// TwinCAT 3 PLC project Xts_Library
// Title: Xts Library
// Company: BeckhoffUK
// Author: ChrisK
// ProjectVersion: 16.0.2
// Description: Xts framework implementation
// ProgramVersion: 3.1.4026.20
// libraries:
//   Base Library, * (Beckhoff UK)
//   Motion Library, * (Beckhoff UK)
//   Tc2_MC2, * (Beckhoff Automation GmbH)
//   Tc2_Standard, * (Beckhoff Automation GmbH)
//   Tc2_System, * (Beckhoff Automation GmbH)
//   Tc3_Mc3Definitions, * (Beckhoff Automation GmbH)
//   Tc3_McCollisionAvoidance, * (Beckhoff Automation GmbH)
//   Tc3_McCoordinatedMotion, * (Beckhoff Automation GmbH)
//   Tc3_Module, * (Beckhoff Automation GmbH)
//   Tc3_XTS_Utility, * (Beckhoff Automation GmbH)
// project tree:
//   Mover Behaviours/ ExtControlBehaviour.TcPOU, StationBehaviour.TcPOU
//   Operations/ Process.TcPOU, Queue.TcPOU, Station.TcPOU, StationSample.TcPOU, Switch.TcPOU, TmsEmbarkStation.TcPOU, TriggerPoint.TcPOU
//   Project Information/ F_GetCompany.TcPOU, F_GetTitle.TcPOU, F_GetVersion.TcPOU
//   Tasks/ XtsDisableSequence.TcPOU, ActivateTrackTask.TcPOU, AddMoverToGroupTask.TcPOU, DisableGroup.TcPOU, EnableGroup.TcPOU, GearCATask.TcPOU, HaltMoverTask.TcPOU, MoveToPositionTask.TcPOU, RemoveAllMoverFromGroup.TcPOU, RemoveMoverFromGroup.TcPOU, ResetGroup.TcPOU, StopMoverGroup.TcPOU, XtsEnableSequence.TcPOU
//   Types/ CAGroupInfo.TcDUT, DisableState.TcDUT (not stored), EmbarkStationStates.TcDUT (not stored), EnableState.TcDUT (not stored), MoverStatus.TcDUT, StationBehaviourInfo.TcDUT (not stored), StationBehaviourState.TcDUT, stStationInfo.TcDUT (not stored), stStationStatus.TcDUT, XtsHardwareInitialisation.TcDUT (not stored), XtsHardwareStatus.TcDUT, XtsPartStatus.TcDUT, XtsSystemInitialisation.TcDUT
//   Interfaces/ IProcess.TcIO, I_CollisionGroup.TcIO, I_ExtControlBehaviour.TcIO, I_Lift.TcIO, I_Station.TcIO (not stored), I_StationBehaviour.TcIO (not stored), I_XTS.TcIO, I_XtsHardware.TcIO, I_XtsIoEnvVar.TcIO, I_XtsMotorModule.TcIO, I_XtsMover.TcIO, I_XtsPart.TcIO, I_XtsTrack.TcIO
//   Mover/ XtsMover.TcPOU
//   / SystemParameters.TcGVL
//   Version/ Global_Version.TcGVL
//   XPU/ XtsIoEnvVar.TcPOU
//   Collision Group/ CollisionGroup.TcPOU
//   Hardware/ NCTController.TcPOU, XTSHardware.TcPOU, XtsMotorModule.TcPOU, XtsPart.TcPOU, XtsTrack.TcPOU
//   XTS/ Xts.TcPOU
// real-time tasks:
//   TASK PlcTask: cycle T#10ms, priority 20, ADS port 350

// ---- Types/CAGroupInfo.TcDUT
TYPE CAGroupInfo :
STRUCT
	sName 		: STRING;
	nId			: OTCID;
	eGroupState	: MC_GROUP_STATE;
	nAxesCount 	: INT; 
END_STRUCT
END_TYPE

// ---- Types/MoverStatus.TcDUT
TYPE MoverStatus :
STRUCT
	isMover1 : BOOL;
	isFrozen : BOOL;
	isLost : BOOL;
	isReadyForPositioning : BOOL;
	isActive : BOOL;
	driveState : DriveState;
	hasControllerError : BOOL32;
END_STRUCT
END_TYPE

// ---- Types/StationBehaviourState.TcDUT
{attribute 'qualified_only'}
{attribute 'strict'}
TYPE StationBehaviourState :
(
	WaitForMoverEnabled := 0,                                               
	WaitingForStart := 1,
	MovingToStart := 2, 
	MoveToFirstStation := 3,                                 
	MovingToCurrentStation := 4,
	ArrivedAtStation := 5,
	MoverQueueingAtStation := 6,
	WaitingForStationComplete := 7,
	StartingProcess := 8,
	MoverInProcess := 9,
	CheckIfFinalStation := 10,
	MovingToNextStation := 11,
	Stopped := 12,
	SequenceError := 99
);
END_TYPE

// ---- Types/stStationStatus.TcDUT
TYPE stStationStatus :
STRUCT
	Empty : BOOL;
	Complete : BOOL;
	Operating : BOOL;
	Ready : BOOL;
	HasMover : BOOL;
END_STRUCT
END_TYPE

// ---- Types/XtsHardwareStatus.TcDUT
TYPE XtsHardwareStatus :
STRUCT
	AllMoversValid : BOOL;
	IsInSim : BOOL;
	ActiveMoverCount : UDINT;
	AreAllModulesInOp : BOOL;
	IsDCLinkVoltageReady : BOOL;
	AreAnyPartsInError : BOOL;
	State : DriveState;
END_STRUCT
END_TYPE

// ---- Types/XtsPartStatus.TcDUT
TYPE XtsPartStatus :
STRUCT
	PartDriveState: Tc3_XTS_Utility.DriveState;
	IsDCLinkReady: BOOL;
	IsPartActive: BOOL;
	PartLength: LREAL;
	AllModuleSsInOP: BOOL;
END_STRUCT
END_TYPE

// ---- Types/XtsSystemInitialisation.TcDUT
{attribute 'qualified_only'}
TYPE XtsSystemInitialisation :
(
	WaitingForXtsIoEnvVar := 0,
	PassGroupReference := 1,
	WaitingForHardwareToInitialise := 2,
	SetATrackForDetection := 3,                                              
	TriggeringRedetection := 4,
	WaitingForAllMoversValid := 5,                                 
	CheckingAllMoverFound := 6,
	CheckIfXtsInSimMode := 7,
	CheckingXts24And48Volts := 8,
	TriggeringMoverIdDetection := 9,
	XtsInitialised := 10,
	InitialisationFault := 99
);
END_TYPE

// ---- SystemParameters.TcGVL
{attribute 'qualified_only'}
VAR_GLOBAL CONSTANT
	NumberOfMovers : UINT := 10;
	NumberOfStations : UINT := 6;
END_VAR

// ---- Version/Global_Version.TcGVL
{attribute 'TcGenerated'}
{attribute 'no-analysis'}
{attribute 'linkalways'}
// This function has been automatically generated from the project information.
VAR_GLOBAL CONSTANT
	{attribute 'const_non_replaced'}
	stLibVersion_Xts_Library : ST_LibVersion := (iMajor := 16, iMinor := 0, iBuild := 2, iRevision := 0, nFlags := 1, sVersion := '16.0.2');
END_VAR

// ---- Interfaces/IProcess.TcIO
INTERFACE IProcess

PROPERTY EndPosition : MC_LREAL
GET
END_GET
END_PROPERTY

PROPERTY ProcessVelocity : mc_lreal
GET
END_GET
END_PROPERTY

END_INTERFACE

// ---- Interfaces/I_CollisionGroup.TcIO
INTERFACE I_CollisionGroup

METHOD AddMoverToThisGroup : HRESULT
VAR_INPUT
	MoverToAdd : I_XtsMover;
END_VAR
END_METHOD

PROPERTY AxisCount : UDINT
GET
END_GET
END_PROPERTY

PROPERTY CAGroupXtsIoEnvInterface : I_Mc2CaGroup
GET
END_GET
SET
END_SET
END_PROPERTY

METHOD Disable : BOOL
VAR_INPUT
END_VAR
END_METHOD

METHOD Enable : BOOL
VAR_INPUT
END_VAR
END_METHOD

PROPERTY ErrorCode : UDINT
GET
END_GET
END_PROPERTY

PROPERTY GroupRef : reference to AXES_GROUP_REF
GET
END_GET
END_PROPERTY

METHOD GroupStop : BOOL
VAR_INPUT
END_VAR
END_METHOD

PROPERTY HasError : BOOL
GET
END_GET
END_PROPERTY

PROPERTY IsDisabled : BOOL
GET
END_GET
END_PROPERTY

PROPERTY IsInErrorStop : BOOL
GET
END_GET
END_PROPERTY

PROPERTY IsInStandBy : BOOL
GET
END_GET
END_PROPERTY

PROPERTY IsMoving : BOOL
GET
END_GET
END_PROPERTY

PROPERTY IsStopping : BOOL
GET
END_GET
END_PROPERTY

PROPERTY MyName : string
GET
END_GET
END_PROPERTY

METHOD RemoveAllMovers : HRESULT
VAR_INPUT
END_VAR
END_METHOD

METHOD RemoveAMover : HRESULT
VAR_INPUT
	MoverToRemove : I_XtsMover;
END_VAR
END_METHOD

METHOD Reset : HRESULT
VAR_INPUT
END_VAR
END_METHOD

END_INTERFACE

// ---- Interfaces/I_ExtControlBehaviour.TcIO
INTERFACE I_ExtControlBehaviour

METHOD Disable : BOOL
VAR_INPUT
END_VAR
END_METHOD

METHOD Enable : BOOL
VAR_INPUT
END_VAR
END_METHOD

METHOD Halt : BOOL
VAR_INPUT
END_VAR
END_METHOD

METHOD MoveTo : BOOL
VAR_INPUT
	Position : LREAL;
	Velocity : LREAL;
END_VAR
END_METHOD

METHOD Reset : BOOL
VAR_INPUT
END_VAR
END_METHOD

END_INTERFACE

// ---- Interfaces/I_Lift.TcIO
INTERFACE I_Lift EXTENDS I_Position

PROPERTY Assigned : BOOL
GET
END_GET
SET
END_SET
END_PROPERTY

METHOD Call : HRESULT
VAR_INPUT
	Position : LREAL;
	Velocity : LREAL;
END_VAR
END_METHOD

END_INTERFACE

// ---- Interfaces/I_XTS.TcIO
INTERFACE I_XTS

METHOD AreAllMoversStationary : BOOL
END_METHOD

METHOD DisableXTS : BOOL
VAR_INPUT
END_VAR
END_METHOD

METHOD EnableXTS : BOOL
VAR_INPUT
END_VAR
END_METHOD

PROPERTY ErrorId : UDINT
GET
END_GET
END_PROPERTY

PROPERTY HasError : BOOL
GET
END_GET
END_PROPERTY

PROPERTY Initialised : BOOL
GET
END_GET
END_PROPERTY

PROPERTY IsIdle : BOOL
GET
END_GET
END_PROPERTY

PROPERTY IsReady : BOOL
GET
END_GET
END_PROPERTY

METHOD PUBLIC Abstract MoverHomeSequence : BOOL
VAR_INPUT
END_VAR
END_METHOD

METHOD RegisterMovers : HRESULT
VAR_INPUT
	MyMover : I_XtsMover;
END_VAR
END_METHOD

METHOD Reset : BOOL
VAR_INPUT
END_VAR
END_METHOD

METHOD StopXts : BOOL
VAR_INPUT
END_VAR
END_METHOD

END_INTERFACE

// ---- Interfaces/I_XtsHardware.TcIO
INTERFACE I_XtsHardware

PROPERTY AllMoverPositionsValid : BOOL
GET
END_GET
END_PROPERTY

PROPERTY AnyPartsInError : BOOL
GET
END_GET
END_PROPERTY

METHOD AreExpectedMoversFound : BOOL
VAR_INPUT
END_VAR
END_METHOD

METHOD CheckTrackSetForDetection : BOOL
VAR_INPUT
	Track : INT;
END_VAR
END_METHOD

PROPERTY ConfiguredDetectionMoverCount : UDINT
GET
END_GET
END_PROPERTY

PROPERTY DetectedNumberOfParts : INT
GET
END_GET
END_PROPERTY

PROPERTY DetectedNumberOfTracks : UINT
GET
END_GET
END_PROPERTY

PROPERTY ExpectedNumberOfParts : int
GET
END_GET
SET
END_SET
END_PROPERTY

PROPERTY ExpectedNumberOfTracks : int
GET
END_GET
SET
END_SET
END_PROPERTY

METHOD GetPartErrorCode : UDINT
END_METHOD

METHOD GetTrackInterfaceByNumber : I_XtsTrack
VAR_INPUT
	TrackNumber : UINT;
END_VAR
END_METHOD

METHOD GetTrackInterfaceByOTCID : I_XtsTrack
VAR_INPUT
	trackOTCID : OTCID;
END_VAR
END_METHOD

METHOD HasValidXPUReference : BOOL
VAR_INPUT
END_VAR
END_METHOD

PROPERTY Initialised : BOOL
GET
END_GET
END_PROPERTY

METHOD IsHardware24VdcOK : HRESULT
VAR_INPUT
END_VAR
END_METHOD

METHOD IsHardware48VdcOK : HRESULT
VAR_INPUT
END_VAR
END_METHOD

METHOD IsIDDetectionStandard : BOOL
VAR_INPUT
END_VAR
END_METHOD

PROPERTY Mover1DetectionState : MoverIdDetectionStateEnum
GET
END_GET
END_PROPERTY

PROPERTY MoverDetectionState : DetectionStateEnum
GET
END_GET
END_PROPERTY

PROPERTY MyName : string
GET
END_GET
END_PROPERTY

PROPERTY MyXpu : I_TcIoXtsProcessingUnit
GET
END_GET
SET
END_SET
END_PROPERTY

PROPERTY MyXts : INT
GET
END_GET
SET
END_SET
END_PROPERTY

PROPERTY NumberOfMoversDetected : UDINT
GET
END_GET
END_PROPERTY

METHOD RemoveATrackFromDetection : HRESULT
VAR_INPUT
	TrackToRemove : UINT;
END_VAR
END_METHOD

METHOD ResetAllParts : BOOL
END_METHOD

METHOD ResetAPart : HRESULT
VAR_INPUT
	Part : UINT;
END_VAR
END_METHOD

METHOD SetATrackForDetection : HRESULT
VAR_INPUT
	TrackToDetect : UINT;
END_VAR
END_METHOD

METHOD SetMoverNumberForDetection : HRESULT
VAR_INPUT
	NumberOfMovers : INT;
END_VAR
END_METHOD

METHOD TriggerMoverDetection : HRESULT
VAR_INPUT
END_VAR
END_METHOD

METHOD TriggerMoverIDDetection : HRESULT
VAR_INPUT
END_VAR
END_METHOD

METHOD TriggerMoverRedetection : HRESULT
VAR_INPUT
END_VAR
END_METHOD

PROPERTY XtsInSim : BOOL
GET
END_GET
END_PROPERTY

END_INTERFACE

// ---- Interfaces/I_XtsIoEnvVar.TcIO
INTERFACE I_XtsIoEnvVar

METHOD GetCaGroupInterface : I_Mc2CaGroup
VAR_INPUT
	CAGroupNumber : INT;
END_VAR
END_METHOD

METHOD GetXPUInterface : I_TcIoXtsProcessingUnit
VAR_INPUT
	MyXts : INT;
END_VAR
END_METHOD

PROPERTY Initialised : BOOL
GET
END_GET
END_PROPERTY

END_INTERFACE

// ---- Interfaces/I_XtsMotorModule.TcIO
INTERFACE I_XtsMotorModule

METHOD AcknowledgeMessages : BOOL
VAR_INPUT
END_VAR
END_METHOD

PROPERTY Act24Vdc : LREAL
GET
END_GET
END_PROPERTY

PROPERTY Act48Vdc : LREAL
GET
END_GET
END_PROPERTY

PROPERTY ControlVdcOK : BOOL
GET
END_GET
END_PROPERTY

PROPERTY MotorVdcOK : BOOL
GET
END_GET
END_PROPERTY

METHOD SetInSim : HRESULT
VAR_INPUT
END_VAR
END_METHOD

END_INTERFACE

// ---- Interfaces/I_XtsMover.TcIO
INTERFACE I_XtsMover

PROPERTY Acceleration : mc_lreal
GET
END_GET
SET
END_SET
END_PROPERTY

METHOD ActivateTrack : HRESULT
VAR_INPUT
	Track : INT;
END_VAR
END_METHOD

METHOD ActivateZeroReferenceSystem : HRESULT
END_METHOD

PROPERTY ActualForce : LREAL
GET
END_GET
END_PROPERTY

PROPERTY ActualPosition : LREAL
GET
END_GET
END_PROPERTY

PROPERTY ActualTrackPosition : LREAL
GET
END_GET
END_PROPERTY

PROPERTY ActualVelocity : LREAL
GET
END_GET
END_PROPERTY

PROPERTY AxisRef : Reference to Axis_ref
GET
END_GET
END_PROPERTY

PROPERTY Deceleration : mc_lreal
GET
END_GET
SET
END_SET
END_PROPERTY

METHOD DisableMover : HRESULT
VAR_INPUT
END_VAR
END_METHOD

METHOD EnableMover : HRESULT
VAR_INPUT
END_VAR
END_METHOD

PROPERTY ErrorID : UDINT
GET
END_GET
END_PROPERTY

PROPERTY Gap : MC_LREAL
GET
END_GET
SET
END_SET
END_PROPERTY

METHOD GetActiveTrackLength : LREAL
VAR_INPUT
END_VAR
END_METHOD

METHOD GetMoverCtrlOTCID : XtsMoverControllerOTCID
VAR_INPUT
END_VAR
END_METHOD

METHOD HaltAxis : HRESULT
VAR_INPUT
END_VAR
END_METHOD

PROPERTY HasError : BOOL
GET
END_GET
END_PROPERTY

PROPERTY PUBLIC IdentInGroup : IDENT_IN_GROUP_REF
GET
END_GET
END_PROPERTY

PROPERTY IsActive : BOOL
GET
END_GET
END_PROPERTY

PROPERTY IsAMover1 : BOOL
GET
END_GET
END_PROPERTY

PROPERTY IsAvoidingCollision : BOOL
GET
END_GET
END_PROPERTY

PROPERTY IsDetected : BOOL
GET
END_GET
END_PROPERTY

PROPERTY IsEnabled : BOOL
GET
END_GET
END_PROPERTY

PROPERTY IsStationary : BOOL
GET
END_GET
END_PROPERTY

PROPERTY Jerk : mc_lreal
GET
END_GET
SET
END_SET
END_PROPERTY

PROPERTY PUBLIC MoversActiveTrack : INT
GET
END_GET
END_PROPERTY

PROPERTY PUBLIC MoverXtsIoEnvInterface : I_TcIoXtsXpuMover
GET
END_GET
SET
END_SET
END_PROPERTY

METHOD MoveTo : HRESULT
VAR_INPUT
	RequiredPosition : MC_LREAL;
	MoveVelocity : MC_LREAL;
	NonModuloMove : BOOL;
END_VAR
END_METHOD

PROPERTY MyCAGroup : I_CollisionGroup
GET
END_GET
SET
END_SET
END_PROPERTY

PROPERTY PositiveDirectionOnly : BOOL
GET
END_GET
SET
END_SET
END_PROPERTY

METHOD RegisterTracks : HRESULT
VAR_INPUT
	Track : I_XtsTrack;
END_VAR
END_METHOD

METHOD Reset : HRESULT
VAR_INPUT
END_VAR
END_METHOD

METHOD SetForceCouple : HRESULT
VAR_INPUT
	XtsMoverCtrlOTCID : Tc3_XTS_Utility.XtsMoverControllerOTCID;
END_VAR
END_METHOD

METHOD SetMoverActiveTrack : HRESULT
VAR_INPUT
	Track : INT;
END_VAR
END_METHOD

METHOD SetParameterSet : HRESULT
VAR_INPUT
	ParameterSet : OTCID;
END_VAR
END_METHOD

METHOD SetSimDetectionPartAndPosition : BOOL
VAR_INPUT
	Part : OTCID;
	Position : LREAL;
END_VAR
END_METHOD

METHOD TriggerMoverArrive : HRESULT
VAR_INPUT
END_VAR
END_METHOD

METHOD TriggerMoverLeave : HRESULT
VAR_INPUT
END_VAR
END_METHOD

END_INTERFACE

// ---- Interfaces/I_XtsPart.TcIO
INTERFACE I_XtsPart

METHOD GetCurrentError : UDINT
VAR_INPUT
END_VAR
END_METHOD

PROPERTY HasError : BOOL
GET
END_GET
END_PROPERTY

METHOD Is24VBusOK : BOOL
END_METHOD

METHOD Is48VBusOK : BOOL
END_METHOD

METHOD ResetPart : BOOL
END_METHOD

METHOD SetInSim : HRESULT
VAR_INPUT
END_VAR
END_METHOD

METHOD SetPartOriginTransform : BOOL
VAR_INPUT
	OriginTransform: Tc3_XTS_Utility.ST_OriginTransform;
END_VAR
END_METHOD

END_INTERFACE

// ---- Interfaces/I_XtsTrack.TcIO
INTERFACE I_XtsTrack

PROPERTY IsTrackSetForDetection : BOOL
GET
END_GET
END_PROPERTY

PROPERTY MyOTCID : OTCID
GET
END_GET
SET
END_SET
END_PROPERTY

METHOD RemoveFromDetection : BOOL
VAR_INPUT
END_VAR
END_METHOD

METHOD SetForDetection : BOOL
VAR_INPUT
END_VAR
END_METHOD

PROPERTY TrackLength : MC_Lreal
GET
END_GET
END_PROPERTY

END_INTERFACE

// ---- Mover Behaviours/ExtControlBehaviour.TcPOU
FUNCTION_BLOCK ExtControlBehaviour IMPLEMENTS I_Cyclic
VAR
	ThisMover : I_XtsMover;
END_VAR

METHOD PUBLIC  Cycle : HRESULT
VAR_INPUT
END_VAR
END_METHOD

METHOD Disable : BOOL
VAR_INPUT
END_VAR
Disable := SUCCEEDED(ThisMover.DisableMover());
END_METHOD

METHOD Enable : BOOL
VAR_INPUT
END_VAR
Enable := SUCCEEDED(ThisMover.EnableMover());
END_METHOD

METHOD Halt : BOOL
VAR_INPUT
END_VAR
Halt := SUCCEEDED(thisMover.HaltAxis());
END_METHOD

METHOD MoveTo : BOOL
VAR_INPUT
	Position : LREAL;
	Velocity : LREAL;
END_VAR
MoveTo := SUCCEEDED(ThisMover.MoveTo(RequiredPosition := Position,
									MoveVelocity := Velocity,
									NonModuloMove := FALSE));
END_METHOD

PROPERTY MyMover : I_XtsMover
GET
MyMover := ThisMover;
END_GET
SET
ThisMover := MyMover;
END_SET
END_PROPERTY

METHOD Reset : BOOL
VAR_INPUT
END_VAR
Reset := SUCCEEDED(ThisMover.Reset());
END_METHOD

END_FUNCTION_BLOCK

// ---- Mover Behaviours/StationBehaviour.TcPOU
FUNCTION_BLOCK StationBehaviour IMPLEMENTS I_Cyclic, I_Resettable, I_Object
VAR
	State : StationBehaviourState;  
	CurrentStation : UINT;
	TargetStationPosition : MC_LREAL;
	_MoverVelocity : MC_LREAL := 1000.0;
	stSequenceInfo : StationBehaviourInfo;
	StationNumber : INT;
	StationArray : ARRAY[0..19] OF I_Station;
	Process : IProcess;
	ThisMover : I_XtsMover;
	ExecuteSequence : BOOL;
	_startPosition : MC_LREAL;
	_XtsNoHome : BOOL;
	_NonModuloMoves : BOOL := FALSE;
END_VAR

{analysis -2}

PROPERTY AbsoluteMoves : bool
GET
AbsoluteMoves := _NonModuloMoves;
END_GET
SET
_NonModuloMoves := AbsoluteMoves;
END_SET
END_PROPERTY

METHOD PUBLIC Cycle : HRESULT
VAR_INPUT
END_VAR
CASE State OF
	StationBehaviourState.WaitForMoverEnabled:
		IF ThisMover.IsEnabled THEN
			State := StationBehaviourState.WaitingForStart;
		END_IF
		
	StationBehaviourState.WaitingForStart:
		IF ExecuteSequence THEN
			State := StationBehaviourState.MovingToStart;
		END_IF
		
	StationBehaviourState.MovingToStart:
		IF (ThisMover.ActualTrackPosition > _startPosition - 0.3 AND ThisMover.ActualTrackPosition < _startPosition + 0.3) OR _XtsNoHome THEN
			State := StationBehaviourState.MoveToFirstStation;
		END_IF
			
	StationBehaviourState.MoveToFirstStation:
		IF StationArray[CurrentStation] <> 0 THEN
			IF SUCCEEDED(ThisMover.MoveTo(RequiredPosition := StationArray[CurrentStation].Position,
								MoveVelocity := _MoverVelocity,
								NonModuloMove := _NonModuloMoves)) THEN
								
				TargetStationPosition := StationArray[CurrentStation].Position;
				State := StationBehaviourState.MovingToCurrentStation;
			END_IF
		END_IF

	StationBehaviourState.MovingToCurrentStation:
		IF ThisMover.IsStationary THEN 
			IF (ThisMover.ActualTrackPosition > TargetStationPosition - 0.3 AND ThisMover.ActualTrackPosition < TargetStationPosition + 0.3) THEN
				State := StationBehaviourState.ArrivedAtStation;
			ELSE
				State := StationBehaviourState.MoverQueueingAtStation;
			END_IF
		END_IF
	
	StationBehaviourState.ArrivedAtStation:
		IF SUCCEEDED(StationArray[CurrentStation].MyMover(ThisMover)) THEN
			IF __QUERYINTERFACE(StationArray[CurrentStation],Process) THEN
				State := StationBehaviourState.StartingProcess;
			ELSE
				State := StationBehaviourState.WaitingForStationComplete;
			END_IF
		END_IF
		
	StationBehaviourState.MoverQueueingAtStation:
		IF NOT ThisMover.IsStationary THEN
				State := StationBehaviourState.MovingToCurrentStation;
		END_IF

	StationBehaviourState.WaitingForStationComplete:
		IF StationArray[CurrentStation].isComplete() THEN
			State := StationBehaviourState.CheckIfFinalStation;
		END_IF

	StationBehaviourState.StartingProcess:
		ThisMover.MoveTo(RequiredPosition := Process.EndPosition,
								MoveVelocity := Process.ProcessVelocity,
								NonModuloMove := _NonModuloMoves);
		State := StationBehaviourState.MoverInProcess;
								
	StationBehaviourState.MoverInProcess:
		IF ThisMover.IsStationary THEN 
			IF (ThisMover.ActualTrackPosition > Process.EndPosition - 0.3 AND ThisMover.ActualTrackPosition < Process.EndPosition + 0.3) THEN
				State := StationBehaviourState.CheckIfFinalStation;
			END_IF
		END_IF
	
	StationBehaviourState.CheckIfFinalStation:
		IF CurrentStation = StationNumber - 1 THEN
			CurrentStation := 0; 
			TargetStationPosition := StationArray[CurrentStation].Position;
			IF SUCCEEDED(ThisMover.MoveTo(RequiredPosition := TargetStationPosition,
							MoveVelocity := _MoverVelocity,
							NonModuloMove := _NonModuloMoves)) THEN
				State := StationBehaviourState.MovingToCurrentStation;
			END_IF
		ELSE
			State := StationBehaviourState.MovingToNextStation;
		END_IF
		
	StationBehaviourState.MovingToNextStation:
		TargetStationPosition := StationArray[CurrentStation + 1].Position;
		IF 	SUCCEEDED(ThisMover.MoveTo(RequiredPosition := TargetStationPosition,
							MoveVelocity := _MoverVelocity,
							NonModuloMove := _NonModuloMoves)) THEN	
			CurrentStation := CurrentStation + 1;
			State := StationBehaviourState.MovingToCurrentStation;
		END_IF	
	StationBehaviourState.Stopped;
		IF ExecuteSequence THEN
			TargetStationPosition := StationArray[CurrentStation].Position;
			IF CurrentStation = 0 THEN
				IF 	SUCCEEDED(ThisMover.MoveTo(RequiredPosition := TargetStationPosition,
									MoveVelocity := _MoverVelocity,
									NonModuloMove := _NonModuloMoves)) THEN	
					State := StationBehaviourState.MovingToCurrentStation;
				END_IF	
			ELSE
				IF 	SUCCEEDED(ThisMover.MoveTo(RequiredPosition := TargetStationPosition,
									MoveVelocity := _MoverVelocity,
									NonModuloMove := _NonModuloMoves)) THEN	
					State := StationBehaviourState.MovingToCurrentStation;
				END_IF	
			END_IF
		END_IF
		
	StationBehaviourState.SequenceError:

	ELSE
		Cycle := E_FAIL;
END_CASE

//Cyclic update info data
stSequenceInfo.CurrentStation := UINT_TO_INT(CurrentStation);
stSequenceInfo.MoverId := ThisMover.AxisRef.NcToPlc.AxisId;
stSequenceInfo.State := State;
stSequenceInfo.Velocity := ThisMover.AxisRef.NcToPlc.ActVelo;
END_METHOD

PROPERTY MoverVelocity : mc_lreal
GET
MoverVelocity := _MoverVelocity;
END_GET
SET
_MoverVelocity := MoverVelocity;
END_SET
END_PROPERTY

PROPERTY MyMover : I_XtsMover
GET
MyMover := ThisMover;
END_GET
SET
ThisMover := MyMover;
END_SET
END_PROPERTY

PROPERTY MyStartPosition : MC_LREAL
GET
MyStartPosition := _startPosition;
END_GET
SET
_startPosition := MyStartPosition;
END_SET
END_PROPERTY

METHOD RegisterAStation : HRESULT
VAR_INPUT
	Station : I_Station;
END_VAR
IF Station = 0 THEN
	RegisterAStation  := -1;
	RETURN;
END_IF
StationArray[StationNumber] := Station;
StationNumber := StationNumber + 1;
END_METHOD

METHOD RegisterWithParent
VAR_INPUT
	Parent	: I_HostObjects;
END_VAR
Parent.RegisterCyclic(THIS^);
END_METHOD

METHOD Reset : HRESULT
VAR_INPUT
END_VAR
State := StationBehaviourState.WaitingForStart;
CurrentStation := 0;
TargetStationPosition := 0.0;
stSequenceInfo.CurrentStation := UINT_TO_INT(CurrentStation);
stSequenceInfo.MoverId := ThisMover.AxisRef.NcToPlc.AxisId;
stSequenceInfo.State := State;
stSequenceInfo.Velocity := ThisMover.AxisRef.NcToPlc.ActVelo;
ExecuteSequence := FALSE;
Reset := 1;
END_METHOD

METHOD StartIndexing : BOOL
VAR_INPUT
END_VAR
ExecuteSequence := TRUE;
END_METHOD

METHOD StopIndexing : BOOL
VAR_INPUT
END_VAR
State := StationBehaviourState.Stopped;
ThisMover.HaltAxis();
END_METHOD

PROPERTY XtsNoHome : BOOL
GET
XtsNoHome := _XtsNoHome;
END_GET
SET
_XtsNoHome := XtsNoHome;
END_SET
END_PROPERTY

END_FUNCTION_BLOCK

// ---- Operations/Process.TcPOU
FUNCTION_BLOCK Process IMPLEMENTS IProcess, I_Station, I_Cyclic, I_Resettable, I_Object
VAR
	_IsClear : BOOL := TRUE;
	_Complete : BOOL;
	_Operating : BOOL;
	_Ready : BOOL := TRUE;
	_Position : LREAL := 0.0;
	_HasMover : BOOL;
	MoverArrive : R_TRIG;
	_MyMover : I_XtsMover;
	_endPos : MC_LREAL;
	_processVelo : MC_LREAL;
	State : INT;
END_VAR

{analysis -2}

METHOD PUBLIC  Cycle : HRESULT
VAR_INPUT
END_VAR
MoverArrive(CLK := _HasMover);
Operation();
IF MoverArrive.Q THEN
	_IsClear := FALSE;
	_Ready := FALSE;
	_Operating := TRUE;
	_Complete := FALSE;
END_IF
END_METHOD

PROPERTY EndPosition : MC_LREAL
GET
EndPosition := _endPos;
END_GET
END_PROPERTY

(*FB_Init is always available implicitly and it is used primarily for initialization.
The return value is not evaluated. For a specific influence, you can also declare the
methods explicitly and provide additional code there with the standard initialization
code. You can evaluate the return value.*)
METHOD FB_Init : BOOL
VAR_INPUT
	(* TRUE: the retain variables are initialized (reset warm / reset cold)*)
	bInitRetains	: BOOL;
	(* TRUE: the instance will be copied to the copy code afterward (online change)   *)
	bInCopyCode	: BOOL;
	Position	: LREAL;
	EndPosition : LREAL;
	ProcessVelocity : LREAL;
END_VAR
_Position := Position;
_endPos := EndPosition;
_processVelo := ProcessVelocity;
END_METHOD

METHOD HasMover : BOOL
VAR_INPUT
END_VAR
HasMover := _HasMover;
END_METHOD

METHOD IsClear : BOOL
IsClear := _IsClear;
END_METHOD

METHOD isComplete : BOOL
isComplete := _Complete;
END_METHOD

METHOD IsOperating : BOOL
IsOperating := _Operating;
END_METHOD

METHOD IsReady : BOOL
IsReady := _Ready;
END_METHOD

METHOD MyMover : HRESULT
VAR_INPUT
	mover : I_XtsMover;
END_VAR
IF mover = 0 THEN
	MyMover := -1;
	RETURN;
END_IF
_HasMover := TRUE;
_MyMover := mover;
END_METHOD

METHOD PROTECTED Operation : BOOL
CASE State OF
	0:
		IF _Operating THEN
			IF Succeeded(_MyMover.MoveTo(RequiredPosition := _endPos,
							MoveVelocity := _processVelo,
							NonModuloMove := FALSE)) THEN
				State := 1;
			END_IF
		END_IF
	1:
		IF _MyMover.ActualTrackPosition = _endPos THEN
			_Operating := FALSE;
			_Complete := TRUE;
			State := 0;
		END_IF
END_CASE	

// IF _Complete AND _HasMover AND_THEN _MyMover.AxisRef.NcToPlc.SetPos > _Position + 50  THEN
// 	_Ready := TRUE;
// 	_HasMover := FALSE;
// 	_IsClear := TRUE;
// 	_MyMover := 0;
// END_IF
END_METHOD

PROPERTY Position : lreal
GET
Position := _Position;
END_GET
END_PROPERTY

PROPERTY ProcessVelocity : MC_LREAL
GET
ProcessVelocity := _processVelo;
END_GET
END_PROPERTY

METHOD RegisterWithParent
VAR_INPUT
	Parent	: I_HostObjects;
END_VAR
Parent.RegisterCyclic(THIS^);
END_METHOD

METHOD Reset : HRESULT
VAR_INPUT
END_VAR
_Complete := FALSE;
_IsClear := TRUE;
_Operating := FALSE;
_Ready := TRUE;
_HasMover := FALSE;
END_METHOD

END_FUNCTION_BLOCK

// ---- Operations/Station.TcPOU
FUNCTION_BLOCK ABSTRACT Station IMPLEMENTS I_Station, I_Cyclic, I_Resettable, I_Object
VAR
	_IsClear : BOOL := TRUE;
	_Complete : BOOL;
	_Operating : BOOL;
	_Ready : BOOL := TRUE;
	_Position : LREAL := 0.0;
	_HasMover : BOOL;
	MoverArrive : R_TRIG;
	_MyMover : I_XtsMover;
END_VAR

{analysis -2}

METHOD PUBLIC  Cycle : HRESULT
VAR_INPUT
END_VAR
MoverArrive(CLK := _HasMover);
Operation();
IF MoverArrive.Q THEN
	_IsClear := FALSE;
	_Ready := FALSE;
	_Operating := TRUE;
	_Complete := FALSE;
END_IF

IF _Complete AND _HasMover AND_THEN _MyMover.AxisRef.NcToPlc.SetPos > _Position + 50  THEN
	_Ready := TRUE;
	_HasMover := FALSE;
	_IsClear := TRUE;
	_MyMover := 0;
END_IF
END_METHOD

//FB_Init is always available implicitly and it is used primarily for initialization.
//The return value is not evaluated. For a specific influence, you can also declare the
//methods explicitly and provide additional code there with the standard initialization
//code. You can evaluate the return value.
METHOD FB_Init: BOOL
VAR_INPUT
    bInitRetains: BOOL; // TRUE: the retain variables are initialized (reset warm / reset cold)
    bInCopyCode: BOOL;  // TRUE: the instance will be copied to the copy code afterward (online change)   
	Position : LREAL;
END_VAR
_Position := Position;
END_METHOD

METHOD HasMover : BOOL
VAR_INPUT
END_VAR
HasMover := _HasMover;
END_METHOD

METHOD IsClear : BOOL
IsClear := _IsClear;
END_METHOD

METHOD isComplete : BOOL
isComplete := _Complete;
END_METHOD

METHOD IsOperating : BOOL
IsOperating := _Operating;
END_METHOD

METHOD IsReady : BOOL
IsReady := _Ready;
END_METHOD

METHOD MyMover : HRESULT
VAR_INPUT
	mover : I_XtsMover;
END_VAR
IF mover = 0 THEN
	MyMover := -1;
	RETURN;
END_IF
IF _HasMover THEN
	MyMover := -2;
	RETURN;
END_IF
_HasMover := TRUE;
_MyMover := mover;
END_METHOD

METHOD PROTECTED ABSTRACT Operation : BOOL
VAR_INPUT
END_VAR
END_METHOD

PROPERTY Position : lreal
GET
Position := _Position;
END_GET
END_PROPERTY

METHOD RegisterWithParent
VAR_INPUT
	Parent	: I_HostObjects;
END_VAR
Parent.RegisterCyclic(THIS^);
END_METHOD

METHOD Reset : HRESULT
VAR_INPUT
END_VAR
_Complete := FALSE;
_IsClear := TRUE;
_Operating := FALSE;
_Ready := TRUE;
_HasMover := FALSE;
END_METHOD

END_FUNCTION_BLOCK

// ---- Operations/Queue.TcPOU
FUNCTION_BLOCK Queue IMPLEMENTS I_Station, I_Cyclic, I_Resettable, I_Object
VAR
	_Position : LREAL := 0.0;
	_MyMover : I_XtsMover;
	_MyLeavingMover : I_XtsMover;
	_NullMover : I_XtsMover;
	_MyStation : I_Station;
	QueueSequence : INT;
	_isComplete : BOOL;
END_VAR

METHOD Cycle : HRESULT
CASE QueueSequence OF
	0:
		IF _MyMover <> 0 AND _MyStation.IsReady() THEN
			_MyLeavingMover := _MyMover;
			_MyMover := 0;
			_isComplete := TRUE;
			QueueSequence := 10;
		END_IF
	10:
		_isComplete := FALSE;
		IF _MyStation.IsOperating() THEN
			_MyLeavingMover := _NullMover;
			QueueSequence := 0;
		END_IF
END_CASE
END_METHOD

//FB_Init is always available implicitly and it is used primarily for initialization.
//The return value is not evaluated. For a specific influence, you can also declare the
//methods explicitly and provide additional code there with the standard initialization
//code. You can evaluate the return value.
METHOD FB_Init: BOOL
VAR_INPUT
    bInitRetains: BOOL; // TRUE: the retain variables are initialized (reset warm / reset cold)
    bInCopyCode: BOOL;  // TRUE: the instance will be copied to the copy code afterward (online change)  
	Position : LREAL; 
	Station : I_Station;
END_VAR
_Position := Position;
_MyStation := Station;
END_METHOD

METHOD HasMover : BOOL
HasMover := _MyMover <> 0;
END_METHOD

METHOD IsClear : BOOL
IsClear := _MyMover = 0;
END_METHOD

METHOD isComplete : BOOL
isComplete := _isComplete;
END_METHOD

METHOD IsOperating : BOOL
IsOperating := _MyMover <> 0;
END_METHOD

METHOD IsReady : BOOL
END_METHOD

METHOD MyMover : HRESULT
VAR_INPUT
	mover	: I_XtsMover;
END_VAR
IF mover = 0 THEN
	MyMover := -1;
	RETURN;
END_IF
IF _MyMover <> 0 THEN
	MyMover := -2;
	RETURN;
END_IF
_MyMover := mover;
END_METHOD

PROPERTY Position : MC_LREAL
GET
Position := _Position;
END_GET
END_PROPERTY

METHOD RegisterWithParent
VAR_INPUT
	Parent	: I_HostObjects;
END_VAR
END_METHOD

METHOD Reset : HRESULT
_isComplete := FALSE;
QueueSequence := 0;
END_METHOD

END_FUNCTION_BLOCK

// ---- Operations/StationSample.TcPOU
FUNCTION_BLOCK StationSample EXTENDS Station
VAR
	_OperationTime : TIME := T#1S;
	DummyOperation : TON;
	State: INT;
END_VAR

{analysis -2}

PROPERTY DummyOperationTime : time
GET
DummyOperationTime := _OperationTime;
END_GET
END_PROPERTY

(*FB_Init is always available implicitly and it is used primarily for initialization.
The return value is not evaluated. For a specific influence, you can also declare the
methods explicitly and provide additional code there with the standard initialization
code. You can evaluate the return value.*)
METHOD FB_Init : BOOL
VAR_INPUT
	(* TRUE: the retain variables are initialized (reset warm / reset cold)*)
	bInitRetains	: BOOL;
	(* TRUE: the instance will be copied to the copy code afterward (online change)   *)
	bInCopyCode	: BOOL;
	Position	: LREAL;
	DummyOperationTime : TIME;
END_VAR
_OperationTime := DummyOperationTime;
END_METHOD

METHOD PROTECTED Operation : BOOL
CASE State OF
	0:
		IF _Operating THEN
			DummyOperation.IN := TRUE;
			State := 1;
		END_IF
	1:
		IF DummyOperation.Q THEN
			_Operating := FALSE;
			_Complete := TRUE;
			DummyOperation.IN := FALSE;
			State := 0;
		END_IF
END_CASE	

DummyOperation(PT := _OperationTime);
END_METHOD

END_FUNCTION_BLOCK

// ---- Operations/Switch.TcPOU
FUNCTION_BLOCK Switch EXTENDS Axis_Base IMPLEMENTS I_Lift
VAR
	_Assigned : BOOL;
END_VAR

PROPERTY Assigned : BOOL
GET
Assigned := _Assigned;
END_GET
SET
_Assigned := Assigned;
END_SET
END_PROPERTY

METHOD Call : HRESULT
VAR_INPUT
	Position : LREAL;
	Velocity : LREAL;
END_VAR
IF Assigned THEN
	RETURN;
	Call := -1;
END_IF

Call := (MoveToPosition(Position := Position, Velocity := Velocity));
END_METHOD

METHOD Release : HRESULT
VAR_INPUT
END_VAR
_Assigned := FALSE;
END_METHOD

END_FUNCTION_BLOCK

// ---- Operations/TmsEmbarkStation.TcPOU
FUNCTION_BLOCK TmsEmbarkStation IMPLEMENTS I_Station, I_Cyclic, I_Resettable, I_Object
VAR
	_IsClear : BOOL := TRUE;
	_Complete : BOOL;
	_Operating : BOOL;
	_Ready : BOOL := TRUE;
	_Position : LREAL := 0.0;
	_HasMover : BOOL;
	MoverArrive : R_TRIG;
	_MyMover : I_XtsMover;
	SwitchAxisPosCtrl : I_Lift;
	_Track1SwitchPosition : MC_LREAL;
	_Track2SwitchPosition : MC_LREAL;
	ExecuteSequence : BOOL;
	_MyTrackNumber : INT := 1;
	_State : EmbarkStationStates;
	_MoverTravelPosition : MC_LREAL;
	_BoardVelocity : MC_LREAL := 100.0;
	_SwitchVelocity : MC_LREAL := 200.0;
	_MoverLeavePosition : LREAL;
	Called : BOOL;
END_VAR

{analysis -2}

PROPERTY BoardVelocity : MC_LREAL
GET
BoardVelocity := _BoardVelocity;
END_GET
SET
_BoardVelocity := BoardVelocity;
END_SET
END_PROPERTY

METHOD Cycle : HRESULT
MoverArrive(CLK := _HasMover);
IF MoverArrive.Q THEN
	_IsClear := FALSE;
	_Ready := FALSE;
	_Operating := TRUE;
	_Complete := FALSE;
END_IF
Operation();
END_METHOD

(*FB_Init is always available implicitly and it is used primarily for initialization.
The return value is not evaluated. For a specific influence, you can also declare the
methods explicitly and provide additional code there with the standard initialization
code. You can evaluate the return value.*)
METHOD FB_Init : BOOL
VAR_INPUT
	(* TRUE: the retain variables are initialized (reset warm / reset cold)*)
	bInitRetains	: BOOL;
	(* TRUE: the instance will be copied to the copy code afterward (online change)   *)
	bInCopyCode	: BOOL;
	Position	: LREAL;
	SwitchAxis : I_Lift;
	MyTrackNumber : INT;
	Track1SwitchPosition : LREAL;
	Track2SwitchPsoition : LREAL;
	MoverOnSwitchPosition : LREAL;
END_VAR
_Position := Position;
SwitchAxisPosCtrl := SwitchAxis;
_MyTrackNumber := MyTrackNumber;
_Track1SwitchPosition := Track1SwitchPosition;
_Track2SwitchPosition := Track2SwitchPsoition;
_MoverTravelPosition := moverOnSwitchPosition;
END_METHOD

METHOD HasMover : BOOL
HasMover := _HasMover;
END_METHOD

METHOD IsClear : BOOL
IsClear := _IsClear;
END_METHOD

METHOD isComplete : BOOL
isComplete := _Complete;
END_METHOD

METHOD IsOperating : BOOL
IsOperating := _Operating;
END_METHOD

METHOD IsReady : BOOL
IsReady := _Ready;
END_METHOD

METHOD MyMover : HRESULT
VAR_INPUT
	mover	: I_XtsMover;
END_VAR
IF mover = 0 THEN
	MyMover := -1;
	RETURN;
END_IF
IF _HasMover THEN
	MyMover := -2;
	RETURN;
END_IF
_HasMover := TRUE;
_MyMover := mover;
END_METHOD

METHOD Operation : BOOL
VAR_INPUT
END_VAR
CASE _State OF
	EmbarkStationStates.Init:
		_Operating := _IsClear := _Complete := _Ready := _HasMover := FALSE;
		_State := EmbarkStationStates.Ready;
	
	EmbarkStationStates.Ready:	
		IF ExecuteSequence THEN
			_Operating := _Complete := _HasMover := FALSE;
			_IsClear := _Ready := TRUE;
			_State := EmbarkStationStates.Waiting;
		END_IF
	
	EmbarkStationStates.Waiting:
		IF _HasMover THEN
			_State := EmbarkStationStates.HasSwitch;
			_Operating := TRUE;
			_IsClear := FALSE;
			_Ready := FALSE;
			_Complete := FALSE;
		END_IF
	
	EmbarkStationStates.HasSwitch:
		IF ((_MyTrackNumber = 1 AND SwitchAxisPosCtrl.isAtPosition(_Track1SwitchPosition))
			OR (_MyTrackNumber = 2 AND SwitchAxisPosCtrl.isAtPosition(_Track2SwitchPosition))) AND NOT SwitchAxisPosCtrl.Assigned THEN
				SwitchAxisPosCtrl.Assigned := TRUE;
				_State := EmbarkStationStates.Boarding;
		ELSIF NOT Called THEN
			_State := EmbarkStationStates.Call;
		END_IF	
		
	EmbarkStationStates.Call:
		IF NOT SwitchAxisPosCtrl.Assigned AND_THEN SwitchAxisPosCtrl.IsStationary() THEN
			IF _MyTrackNumber = 1 THEN
				SwitchAxisPosCtrl.Call(Position := _Track1SwitchPosition, Velocity := _SwitchVelocity);
			ELSE
				SwitchAxisPosCtrl.Call(Position := _Track2SwitchPosition, Velocity := _SwitchVelocity);
			END_IF
			SwitchAxisPosCtrl.Assigned := TRUE;
			Called := TRUE;
			_State := EmbarkStationStates.test;
		END_IF
		
	EmbarkStationStates.test:
		IF (_MyTrackNumber = 1 AND SwitchAxisPosCtrl.isAtPosition(_Track1SwitchPosition))
			OR (_MyTrackNumber = 2 AND SwitchAxisPosCtrl.isAtPosition(_Track2SwitchPosition)) THEN
				_State := EmbarkStationStates.Boarding;
				Called := FALSE;
		END_IF	
		
	EmbarkStationStates.Boarding:
		_MyMover.MoveTo(RequiredPosition := _MoverTravelPosition, MoveVelocity := _BoardVelocity, NonModuloMove := FALSE);
		IF _MoverTravelPosition > _MyMover.GetActiveTrackLength() THEN
			IF (_MyMover.ActualTrackPosition > (_MoverTravelPosition - _MyMover.GetActiveTrackLength()) - 0.3 
				AND _MyMover.ActualTrackPosition < (_MoverTravelPosition - _MyMover.GetActiveTrackLength()) + 0.3) THEN
				_State := EmbarkStationStates.BoardingComplete;
			END_IF
		ELSE
			IF (_MyMover.ActualTrackPosition > _MoverTravelPosition - 0.3 AND _MyMover.ActualTrackPosition < _MoverTravelPosition + 0.3) THEN
				_State := EmbarkStationStates.BoardingComplete;
			END_IF
		END_IF
		
	EmbarkStationStates.BoardingComplete:
		IF _MyTrackNumber = 1 THEN
			SwitchAxisPosCtrl.MoveToPosition(Position := _Track2SwitchPosition, Velocity := _SwitchVelocity);
		ELSE
			SwitchAxisPosCtrl.MoveToPosition(Position := _Track1SwitchPosition, Velocity := _SwitchVelocity);
		END_IF
		_State := EmbarkStationStates.Moving;
		
	EmbarkStationStates.Moving:
		IF (_MyTrackNumber = 1 AND SwitchAxisPosCtrl.isAtPosition(position := _Track2SwitchPosition)) OR
			(_MyTrackNumber = 2 AND SwitchAxisPosCtrl.isAtPosition(position := _Track1SwitchPosition)) THEN
			_State := EmbarkStationStates.ActivateTrackForMover;
		END_IF
		
	EmbarkStationStates.ActivateTrackForMover:
		IF _MyTrackNumber = 1 THEN
			IF SUCCEEDED(_MyMover.ActivateTrack(Track := 2)) THEN
				_State := EmbarkStationStates.CheckActiveTrack;
			END_IF
		ELSE
			IF SUCCEEDED(_MyMover.ActivateTrack(Track := 1)) THEN
				_State := EmbarkStationStates.CheckActiveTrack;
			END_IF
		END_IF
		
	EmbarkStationStates.CheckActiveTrack:
		IF _MyTrackNumber = 1 AND_THEN _MyMover.MoversActiveTrack = 2 THEN
			_State := EmbarkStationStates.CheckMoverLeft;
			_MoverLeavePosition := _MyMover.AxisRef.NcToPlc.ActPos;
		ELSIF  _MyMover.MoversActiveTrack = 1 THEN
			_State := EmbarkStationStates.CheckMoverLeft;
			_MoverLeavePosition := _MyMover.AxisRef.NcToPlc.ActPos;
		END_IF
	
	EmbarkStationStates.CheckMoverLeft:
		_Complete := TRUE;
		IF _MyMover.AxisRef.NcToPlc.ActPos > _MoverLeavePosition + 100 THEN
			_State := EmbarkStationStates.Done;
			_HasMover := FALSE;
			SwitchAxisPosCtrl.Assigned := FALSE;
		END_IF
			
	EmbarkStationStates.Done:
		IF _Complete AND NOT _HasMover THEN
			_Operating := FALSE;
			_IsClear := TRUE;
			_Ready := TRUE;
			_State := EmbarkStationStates.Waiting;
		END_IF	
END_CASE
END_METHOD

PROPERTY Position : MC_LREAL
GET
Position := _Position;
END_GET
END_PROPERTY

METHOD RegisterWithParent
VAR_INPUT
	Parent	: Base_Library.I_HostObjects;
END_VAR
END_METHOD

METHOD Reset : HRESULT
_Complete := FALSE;
_IsClear := TRUE;
_Operating := FALSE;
_Ready := TRUE;
_HasMover := FALSE;
_State := EmbarkStationStates.Init;
SwitchAxisPosCtrl.Assigned := FALSE;
END_METHOD

METHOD StartSwitch : BOOL
VAR_INPUT
END_VAR
ExecuteSequence := TRUE;
END_METHOD

METHOD StopSwitch : BOOL
VAR_INPUT
END_VAR
ExecuteSequence := FALSE;
END_METHOD

PROPERTY SwitchVelocity : LREAL
GET
SwitchVelocity := _SwitchVelocity;
END_GET
SET
_SwitchVelocity := SwitchVelocity;
END_SET
END_PROPERTY

END_FUNCTION_BLOCK

// ---- Operations/TriggerPoint.TcPOU
FUNCTION_BLOCK TriggerPoint IMPLEMENTS I_Cyclic, I_Resettable, I_Object
VAR
	_TriggerPointMovers : ARRAY[0..MaxMovers] OF I_XtsMover;
	SystemMovers : ARRAY[0..MaxMovers] OF I_XtsMover;
	NumberOfMovers : INT;
	_position : LREAL;
	_range : LREAL;
END_VAR
VAR CONSTANT
	MaxMovers : INT := 10;
END_VAR

METHOD Cycle : HRESULT
VAR 
	i : INT;
	arrivingMover : I_XtsMover;
	detected : BOOL;
END_VAR
FOR i := 0 TO MaxMovers DO
	IF SystemMovers[i] <> 0 THEN
		IF SystemMovers[i].AxisRef.NcToPlc.ModuloActPos < _position + 10.0 AND
			SystemMovers[i].AxisRef.NcToPlc.ModuloActPos > _position - 10.0 THEN
			arrivingMover := SystemMovers[i];
		END_IF
	END_IF
END_FOR
IF arrivingMover <> 0 THEN
	FOR i := 0 TO MaxMovers DO
		IF arrivingMover = _TriggerPointMovers[i] THEN
			detected := TRUE;
		END_IF
	END_FOR
	IF NOT detected THEN
		FOR i := 0 TO MaxMovers DO
			IF _TriggerPointMovers[i] = 0 THEN
				_TriggerPointMovers[i] := arrivingMover;
				EXIT;
			END_IF
		END_FOR
	END_IF
END_IF
FOR i := 0 TO MaxMovers DO
	IF _TriggerPointMovers[i] <> 0 AND_THEN 
		_TriggerPointMovers[i].AxisRef.NcToPlc.ModuloActPos > _position + _range THEN
		_TriggerPointMovers[i] := 0;
	END_IF
END_FOR
END_METHOD

//FB_Init is always available implicitly and it is used primarily for initialization.
//The return value is not evaluated. For a specific influence, you can also declare the
//methods explicitly and provide additional code there with the standard initialization
//code. You can evaluate the return value.
METHOD FB_Init: BOOL
VAR_INPUT
    bInitRetains: BOOL; // TRUE: the retain variables are initialized (reset warm / reset cold)
    bInCopyCode: BOOL;  // TRUE: the instance will be copied to the copy code afterward (online change)   
	Position : LREAL;
	Range : LREAL;
END_VAR
_range := Range;
_position := Position;
END_METHOD

PROPERTY Position : lreal
GET
Position := _Position;
END_GET
END_PROPERTY

METHOD RegisterMovers : HRESULT
VAR_INPUT
	MyMover : I_XtsMover;
END_VAR
VAR
	i : uINT;
END_VAR
IF MyMover <> 0 THEN
	SystemMovers[NumberOfMovers] := MyMover;
	NumberOfMovers := NumberOfMovers + 1;
ELSE
	RegisterMovers := -1;
END_IF
END_METHOD

METHOD RegisterWithParent
VAR_INPUT
	Parent	: Base_Library.I_HostObjects;
END_VAR
END_METHOD

METHOD Reset : HRESULT
VAR
	i : INT;
END_VAR
FOR i := 0 TO MaxMovers DO
	_TriggerPointMovers[i] := 0;
END_FOR
END_METHOD

END_FUNCTION_BLOCK

// ---- Project Information/F_GetCompany.TcPOU
// This function has been automatically generated from the project information.
{attribute 'signature_flag' := '1073741824'}
{attribute 'TcGenerated'}
{attribute 'no-analysis'}
FUNCTION F_GetCompany : WSTRING
VAR_INPUT
	
END_VAR

F_GetCompany := "BeckhoffUK";

END_FUNCTION

// ---- Project Information/F_GetTitle.TcPOU
// This function has been automatically generated from the project information.
{attribute 'signature_flag' := '1073741824'}
{attribute 'TcGenerated'}
{attribute 'no-analysis'}
FUNCTION F_GetTitle : WSTRING
VAR_INPUT
	
END_VAR

F_GetTitle := "Xts Library";

END_FUNCTION

// ---- XTS/Xts.TcPOU
FUNCTION_BLOCK ABSTRACT Xts IMPLEMENTS I_Cyclic, I_Initialisable, I_XTS, I_Object
VAR
	MyName : STRING;
	_MyXts : INT;
	_XtsEnabled : BOOL;
	_XPU : I_TcIoXtsProcessingUnit;
	_MoverArray : ARRAY[0..MaxMovers] OF I_XtsMover;
	_XtsIoEnvVar : I_XtsIoEnvVar;
	ICollisionGroup : I_CollisionGroup;
	_MyXtsHardware : I_XtsHardware;
	XtsHwState : XtsSystemInitialisation;
	EnableSequence : XtsEnableSequence;
	DisableSequence : XtsDisableSequence;	
	_Initialised : BOOL;
	EnabledTrigger : R_TRIG;
	DisabledTrigger : R_TRIG;
	_registeredNumberOfMovers: INT;
	DetectedMoverCount : UDINT;
	HardwareError : BOOL;
	CAGroupError : BOOL;
	_ErrorID : UDINT;
END_VAR
VAR CONSTANT
	MaxMovers : INT := 255;
END_VAR

{analysis -2}

METHOD AreAllMoversStationary : BOOL
VAR
	i : INT;
END_VAR
AreAllMoversStationary := TRUE;
FOR i := 0 TO _registeredNumberOfMovers - 1 DO
	IF NOT _MoverArray[i].IsStationary THEN
		AreAllMoversStationary := FALSE;
		EXIT;
	END_IF
END_FOR
END_METHOD

METHOD PUBLIC Cycle : HRESULT
VAR
	EnableResult : HRESULT;
	DisableResult : HRESULT;
	GrpStopResult : HRESULT;
	CollisionResult : HRESULT;
END_VAR
IF NOT _Initialised THEN	
	Cycle  := -1;
	RETURN;
END_IF

EnableResult := EnableSequence.Cycle();
DisableResult := DisableSequence.Cycle();
EnabledTrigger(CLK := EnableSequence.Done);
DisabledTrigger(CLK := DisableSequence.Done);
IF EnabledTrigger.Q THEN
	_XtsEnabled := TRUE;
END_IF
IF DisabledTrigger.Q THEN
	_XtsEnabled := false;
END_IF

HardwareError := _MyXtsHardware.AnyPartsInError;
CAGroupError := ICollisionGroup.HasError;

IF CAGroupError THEN
	_ErrorID := ICollisionGroup.ErrorCode;
END_IF
IF HardwareError THEN
	_ErrorID := _MyXtsHardware.GetPartErrorCode();
END_IF
IF NOT CAGroupError AND NOT HardwareError THEN
	_ErrorID := 0;
END_IF
END_METHOD

METHOD DisableXTS : BOOL
VAR_INPUT
END_VAR
IF _XtsEnabled THEN
	Base_Library.Tracing.Trace.Verbose(MyName, 'Disable Accepted');
	DisableXTS := SUCCEEDED(DisableSequence.Disable());
END_IF
END_METHOD

METHOD EnableXTS : BOOL
VAR_INPUT
END_VAR
IF NOT _XtsEnabled THEN
	Base_Library.Tracing.Trace.Verbose(MyName, 'Enable Accepted');
	EnableXts := SUCCEEDED(EnableSequence.Enable());
END_IF
END_METHOD

PROPERTY ErrorId : UDINT
GET
_ErrorID := _ErrorID;
END_GET
END_PROPERTY

PROPERTY ExpectedNumberOfParts : int
GET
ExpectedNumberOfParts := _MyXtsHardware.ExpectedNumberOfParts;
END_GET
SET
_MyXtsHardware.ExpectedNumberOfParts := ExpectedNumberOfParts;
END_SET
END_PROPERTY

PROPERTY ExpectedNumberOfTracks : int
GET
ExpectedNumberOfTracks := _MyXtsHardware.ExpectedNumberOfTracks;
END_GET
SET
_MyXtsHardware.ExpectedNumberOfTracks := ExpectedNumberOfTracks;
END_SET
END_PROPERTY

//FB_Init is always available implicitly and it is used primarily for initialization.
//The return value is not evaluated. For a specific influence, you can also declare the
//methods explicitly and provide additional code there with the standard initialization
//code. You can evaluate the return value.
METHOD FB_Init: BOOL
VAR_INPUT
    bInitRetains: BOOL; // TRUE: the retain variables are initialized (reset warm / reset cold)
    bInCopyCode: BOOL;  // TRUE: the instance will be copied to the copy code afterward (online change)   
	MyXtsIoEnvVar : I_XtsIoEnvVar;
	MyXtsHardware : I_XtsHardware;
	MyCAGroup : I_CollisionGroup;
END_VAR
_XtsIoEnvVar := MyXtsIoEnvVar;
_MyXtsHardware := MyXtsHardware;
ICollisionGroup := MyCAGroup;
EnableSequence.MyCollisionGroup := ICollisionGroup;
DisableSequence.MyCollisionGroup := ICollisionGroup;
END_METHOD

PROPERTY HasError : BOOL
GET
HasError := ICollisionGroup.HasError OR _MyXtsHardware.AnyPartsInError;
END_GET
END_PROPERTY

METHOD Initialise : HRESULT
VAR
	i : INT;
END_VAR
Initialise := -1;
CASE XtsHwState OF
	XtsSystemInitialisation.WaitingForXtsIoEnvVar:
		IF _XtsIoEnvVar.Initialised THEN
			_XPU := _XtsIoEnvVar.GetXPUInterface(_MyXts);
			_MyXtsHardware.MyXpu := _XPU;
			XtsHwState := XtsSystemInitialisation.PassGroupReference;
		END_IF
		
	XtsSystemInitialisation.PassGroupReference:
		ICollisionGroup.CAGroupXtsIoEnvInterface := _XtsIoEnvVar.GetCaGroupInterface(_MyXts);
		XtsHwState := XtsSystemInitialisation.WaitingForHardwareToInitialise;
	
	XtsSystemInitialisation.WaitingForHardwareToInitialise:
		IF _MyXtsHardware.Initialised THEN
			MyName := _MyXtsHardware.MyName;
			XtsHwState := XtsSystemInitialisation.SetATrackForDetection;
		END_IF
	
	XtsSystemInitialisation.SetATrackForDetection:
		IF SUCCEEDED(_MyXtsHardware.SetATrackForDetection(1)) THEN
			XtsHwState := XtsSystemInitialisation.TriggeringRedetection;
		END_IF
		
	XtsSystemInitialisation.TriggeringRedetection:
		IF SUCCEEDED(_MyXtsHardware.TriggerMoverRedetection()) THEN
			XtsHwState := XtsSystemInitialisation.WaitingForAllMoversValid;
		END_IF
		
	XtsSystemInitialisation.WaitingForAllMoversValid:
		IF _MyXtsHardware.AllMoverPositionsValid THEN
			XtsHwState := XtsSystemInitialisation.CheckingAllMoverFound;
		END_IF
	
	XtsSystemInitialisation.CheckingAllMoverFound:
		IF _MyXtsHardware.AreExpectedMoversFound() THEN
			DetectedMoverCount := _MyXtsHardware.NumberOfMoversDetected;
			XtsHwState := XtsSystemInitialisation.CheckIfXtsInSimMode;
		END_IF
		
	XtsSystemInitialisation.CheckIfXtsInSimMode:
		IF _MyXtsHardware.XtsInSim THEN
			XtsHwState := XtsSystemInitialisation.TriggeringMoverIdDetection;
		ELSE
			XtsHwState := XtsSystemInitialisation.CheckingXts24And48Volts;
		END_IF
		
	XtsSystemInitialisation.CheckingXts24And48Volts:
		IF SUCCEEDED(_MyXtsHardware.IsHardware24VdcOK()) AND SUCCEEDED(_MyXtsHardware.IsHardware48VdcOK()) THEN
			XtsHwState := XtsSystemInitialisation.TriggeringMoverIdDetection;
		END_IF
	
	XtsSystemInitialisation.TriggeringMoverIdDetection:
		IF _MyXtsHardware.IsIDDetectionStandard() OR_ELSE SUCCEEDED(_MyXtsHardware.TriggerMoverIDDetection()) THEN
			XtsHwState := XtsSystemInitialisation.XtsInitialised;
		END_IF
	
	XtsSystemInitialisation.XtsInitialised:
		Initialise := 0;
		_Initialised := TRUE;	
END_CASE
END_METHOD

PROPERTY Initialised : BOOL
GET
Initialised := _Initialised;
END_GET
END_PROPERTY

PROPERTY IsIdle : BOOL
GET
IsIdle := DisableSequence.Done;
END_GET
END_PROPERTY

PROPERTY IsReady : BOOL
GET
IsReady := _XtsEnabled;
END_GET
END_PROPERTY

METHOD PUBLIC Abstract MoverHomeSequence : BOOL
VAR_INPUT
END_VAR
END_METHOD

PROPERTY MyXts : INT
GET
MyXts := _MyXtsHardware.MyXts;
END_GET
SET
_MyXtsHardware.MyXts := _MyXts := MyXts;
END_SET
END_PROPERTY

METHOD RegisterMovers : HRESULT
VAR_INPUT
	MyMover : I_XtsMover;
END_VAR
VAR
	i : UINT;
	MoverRegistered: BOOL;
END_VAR
IF MyMover = 0 THEN
	Base_Library.Tracing.Trace.Warning(MyName, 'Register Mover Fail - null ptr');
	RegisterMovers := -1;
	RETURN;
END_IF
IF NOT _Initialised THEN
	Base_Library.Tracing.Trace.Warning(MyName, 'Register Mover Fail - not ready');
	RegisterMovers := -2;
	RETURN;
END_IF
IF _registeredNumberOfMovers >= MaxMovers THEN
	Base_Library.Tracing.Trace.Warning(MyName, 'Register Mover Fail - max movers reached');
	RegisterMovers := -3;
	RETURN;
END_IF
FOR i := 0 TO (_registeredNumberOfMovers - 1) DO
	IF _MoverArray[i] = MyMover THEN
		MoverRegistered := TRUE;
		EXIT;
	END_IF
END_FOR
IF MoverRegistered THEN
	Base_Library.Tracing.Trace.Warning(MyName, 'Register Mover Fail - registered');
	RegisterMovers := -4;
	RETURN;
END_IF

Base_Library.Tracing.Trace.Verbose(MyName, 'Register Mover Accepted');
_MoverArray[_registeredNumberOfMovers] := MyMover;
_registeredNumberOfMovers := _registeredNumberOfMovers + 1;
EnableSequence.RegisterMovers(MyMover);
DisableSequence.RegisterMovers(MyMover);
FOR i := 1 TO _MyXtsHardware.DetectedNumberOfTracks DO
	MyMover.RegisterTracks(Track := _MyXtsHardware.GetTrackInterfaceByNumber(i));
END_FOR
FOR i := 1 TO TO_UINT(_XPU.GetDetectedMoverCount()) DO
	IF MyMover.AxisRef.NcToPlc.AxisId = _XPU.MoverTcIo(i).P_AxisId THEN
		MyMover.MoverXtsIoEnvInterface := _XPU.MoverTcIo(i);
	END_IF
END_FOR
END_METHOD

METHOD RegisterWithParent
VAR_INPUT
	Parent	: I_HostObjects;
END_VAR
Parent.RegisterCyclic(THIS^);
Parent.RegisterInitialisable(THIS^);
END_METHOD

METHOD Reset : BOOL
VAR_INPUT
END_VAR
Reset := SUCCEEDED(ICollisionGroup.Reset());
_MyXtsHardware.ResetAllParts();
Base_Library.Tracing.Trace.Verbose(MyName, 'Reset Accepted');
END_METHOD

METHOD StopXts : BOOL
VAR_INPUT
END_VAR
StopXTS := ICollisionGroup.GroupStop();
Base_Library.Tracing.Trace.Verbose(MyName, 'Stop Accepted');
END_METHOD

END_FUNCTION_BLOCK

// ---- Tasks/XtsEnableSequence.TcPOU
FUNCTION_BLOCK XtsEnableSequence  IMPLEMENTS I_Task
VAR
	_caGroup : I_CollisionGroup;
	moverIndex : UINT;
	AllMoversEnabled: BOOL;
	EnableTrigger : BOOL;	
	arrMovers : ARRAY[0..MaxMovers] OF I_XtsMover;
	_registeredNumberOfMovers : INT;
	State: EnableState;
	_Done: BOOL;
	_Error: BOOL;
	_Busy: BOOL;
END_VAR
VAR CONSTANT
	MaxMovers : INT := 255;
END_VAR

{analysis -2}

METHOD Abort : BOOL
EnableTrigger := FALSE;
State := 0;
END_METHOD

PROPERTY Busy : BOOL
GET
Busy := _Busy;
END_GET
END_PROPERTY

METHOD Cycle : HRESULT
VAR
	i : INT;
END_VAR
CASE State OF
	EnableState.Idle:
		IF EnableTrigger THEN
			Cycle := S_PENDING;
			State := EnableState.Reset_Movers;
			EnableTrigger := FALSE;
			moverIndex := 0;
			_Busy := TRUE;
			_Done := FALSE;
			_Error := FALSE;
		END_IF
		
	EnableState.Reset_Movers:
		FOR i := 0 TO (_registeredNumberOfMovers-1) DO
			arrMovers[i].Reset();
		END_FOR
		State := EnableState.Reset_Group;
		
	EnableState.Reset_Group:
		IF _caGroup.IsInErrorStop THEN
			_caGroup.Reset();
		END_IF
		State := EnableState.Add_Mover;
		
	EnableState.Add_Mover:
		IF Succeeded( _caGroup.AddMoverToThisGroup(MoverToAdd := arrMovers[moverIndex])) THEN
			State := EnableState.Check_Add_Mover;
		END_IF
		
		
	EnableState.Check_Add_Mover:
		IF moverIndex <> (_registeredNumberOfMovers-1) THEN
			moverIndex := moverIndex + 1;
			State := EnableState.Add_Mover;
		ELSE
			FOR i := 0 TO (_registeredNumberOfMovers-1) DO
				arrMovers[i].EnableMover();
			END_FOR
			State := EnableState.Enable_Movers;
		END_IF
		
	EnableState.Enable_Movers:
		AllMoversEnabled := TRUE;
		FOR i := 0 TO (_registeredNumberOfMovers-1) DO
			AllMoversEnabled := TRUE AND arrMovers[i].IsEnabled;
		END_FOR
		IF AllMoversEnabled THEN
			
			State := EnableState.Enable_Group;
		END_IF

	EnableState.Enable_Group:
		IF _caGroup.Enable() THEN
			State := EnableState.Check_Standby;
		END_IF
		
	EnableState.Check_Standby:
		IF _caGroup.IsInStandBy THEN
			State := EnableState.Idle;
			_Busy := FALSE;
			_Done := TRUE;
			Cycle := S_OK;
		END_IF
	ELSE
		Cycle := E_FAIL;
		_Busy := FALSE;
		_Done := FALSE;
		_Error := TRUE;
END_CASE
END_METHOD

PROPERTY Done : BOOL
GET
Done := _Done;
END_GET
END_PROPERTY

METHOD Enable : HRESULT
VAR_INPUT
END_VAR
IF _registeredNumberOfMovers = 0 THEN
	Enable := -1;
	RETURN;
END_IF

IF EnableTrigger THEN
	Enable := -2;
	RETURN;
END_IF

IF _caGroup = 0 THEN
	Enable := -3;
	RETURN;
END_IF

EnableTrigger := TRUE;
END_METHOD

PROPERTY Error : BOOL
GET
Error := _Error;
END_GET
END_PROPERTY

PROPERTY MyCollisionGroup : I_CollisionGroup
GET
MyCollisionGroup := _caGroup;
END_GET
SET
IF MyCollisionGroup <> 0 THEN
	_caGroup := MyCollisionGroup;
END_IF
END_SET
END_PROPERTY

PROPERTY RegisteredMoverNumber : INT
GET
RegisteredMoverNumber := _registeredNumberOfMovers;
END_GET
END_PROPERTY

METHOD RegisterMovers : HRESULT
VAR_INPUT
	MyMover : I_XtsMover;
END_VAR
IF MyMover = 0 THEN
	RegisterMovers := -1;
	RETURN;
END_IF

arrMovers[_registeredNumberOfMovers] := MyMover;
_registeredNumberOfMovers := _registeredNumberOfMovers + 1;
END_METHOD

END_FUNCTION_BLOCK

// ---- Tasks/XtsDisableSequence.TcPOU
FUNCTION_BLOCK XtsDisableSequence IMPLEMENTS I_Task
VAR
	_caGroup : I_CollisionGroup;
	DisableTrigger: BOOL;
	moverNumbers : UINT := 1;
	AllMoversDisabled: BOOL;	
	arrMovers : ARRAY[0..MaxMovers] OF I_XtsMover;
	_registeredNumberOfMovers : INT;
	CaGroupResetResult: BOOL;
	State: DisableState;
	_Done: BOOL;
	_Error: BOOL;
	_Busy: BOOL;
END_VAR
VAR CONSTANT
	MaxMovers : INT := 255;
END_VAR

{analysis -2}

METHOD Abort : BOOL
VAR
END_VAR
DisableTrigger := FALSE;
State := 0;
Abort := true;
END_METHOD

PROPERTY Busy : BOOL
GET
Busy := _Busy;
END_GET
END_PROPERTY

METHOD Cycle : HRESULT
VAR
	i : INT;
END_VAR
CASE State OF
	DisableState.Idle:
		IF DisableTrigger THEN
			Cycle := S_PENDING;
			DisableTrigger := FALSE;
			_Busy := TRUE;
			_Done := FALSE;
			_Error := FALSE;
			State := DisableState.Group_Stop;
		END_IF
		
	DisableState.Group_Stop:
		IF _caGroup.IsMoving THEN
			_caGroup.GroupStop();
		END_IF
		State := DisableState.Remove_Movers;
		
	DisableState.Remove_Movers:
		IF _caGroup.IsInStandBy THEN
			IF SUCCEEDED(_caGroup.RemoveAllMovers()) THEN
				State := DisableState.Disable_Movers;
			END_IF
		END_IF
	
	DisableState.Disable_Movers:
		IF _caGroup.AxisCount = 0 THEN
			FOR i := 0 TO (_registeredNumberOfMovers-1) DO
				arrMovers[i].DisableMover();
			END_FOR
			State := DisableState.Disable_Group;
		END_IF
		
	DisableState.Disable_Group:
		AllMoversDisabled := TRUE;
		FOR i := 0 TO (_registeredNumberOfMovers-1) DO
			AllMoversDisabled := AllMoversDisabled AND NOT arrMovers[i].IsEnabled;
		END_FOR
		IF AllMoversDisabled THEN
			State := DisableState.Reset_Group;
			_caGroup.Disable();
		END_IF
		
	DisableState.Reset_Group:
		IF _caGroup.IsInErrorStop THEN
			_caGroup.Reset();
		END_IF	
		State := DisableState.Wait_For_Disabled;
		
	DisableState.Wait_For_Disabled:
		IF _caGroup.IsDisabled THEN
			State := DisableState.Idle;
			Cycle := S_OK;
			_Busy := FALSE;
			_Done := TRUE;
		END_IF
	ELSE
		Cycle := E_FAIL;
		_Busy := FALSE;
		_Done := FALSE;
		_Error := TRUE;
END_CASE
END_METHOD

METHOD Disable : HRESULT
VAR_INPUT
END_VAR
IF _registeredNumberOfMovers = 0 THEN
	Disable := -1;
	RETURN;
END_IF

IF DisableTrigger THEN
	Disable := -2;
	RETURN;
END_IF

IF _caGroup = 0 THEN
	Disable := -3;
	RETURN;
END_IF

DisableTrigger := TRUE;
END_METHOD

PROPERTY Done : BOOL
GET
Done := _Done;
END_GET
END_PROPERTY

PROPERTY Error : BOOL
GET
Error := _Error;
END_GET
END_PROPERTY

PROPERTY MyCollisionGroup : I_CollisionGroup
GET
MyCollisionGroup := _caGroup;
END_GET
SET
IF MyCollisionGroup <> 0 THEN
	_caGroup := MyCollisionGroup;
END_IF
END_SET
END_PROPERTY

PROPERTY RegisteredMoverNumber : INT
GET
RegisteredMoverNumber := _registeredNumberOfMovers;
END_GET
END_PROPERTY

METHOD RegisterMovers : HRESULT
VAR_INPUT
	MyMover : I_XtsMover;
END_VAR
IF MyMover = 0 THEN
	RegisterMovers := -1;
	RETURN;
END_IF

arrMovers[_registeredNumberOfMovers] := MyMover;
_registeredNumberOfMovers := _registeredNumberOfMovers + 1;
END_METHOD

END_FUNCTION_BLOCK

// ---- Project Information/F_GetVersion.TcPOU
// This function has been automatically generated from the project information.
{attribute 'signature_flag' := '1073741824'}
{attribute 'TcGenerated'}
{attribute 'no-analysis'}
FUNCTION F_GetVersion : ST_LibVersion
VAR_INPUT
	
END_VAR

F_GetVersion.iMajor := 16;
F_GetVersion.iMinor := 0;
F_GetVersion.iBuild := 2;
F_GetVersion.iRevision := 0;
F_GetVersion.sVersion := '16.0.2';
F_GetVersion.nFlags := 1;

END_FUNCTION

// ---- Mover/XtsMover.TcPOU
FUNCTION_BLOCK XtsMover IMPLEMENTS I_Cyclic, I_XtsMover, I_Resettable, I_Object
VAR
	MyAxisRef : AXIS_REF;
	_MyAxisStatus : ST_AxisStatus;
	_MyNCData : NCTOPLC_AXIS_REF;
	TaskCollection : ObjectRunner<99>;
	EnableBehaviour : EnableDisableTask := (AxisRef := MyAxisRef);
	MoveBehaviour : MoveToPositionTask:= (AxisRef := MyAxisRef);
	HaltBehaviour : HaltMoverTask := (AxisRef := MyAxisRef);
	ResetBehaviour : CoEResetTask := (AxisRef := MyAxisRef);
	MoverActivateTrackBehaviour : ActivateTrackTask:= (AxisRef := MyAxisRef);
	_ipTcIoXtsMover	: I_TcIoXtsXpuMover;
	TrackChangeTrigger : R_TRIG;
	_MoverAbsMoveOptions : ST_MoveAbsoluteCAOptions;
	_stTmsActPositions : ST_PositionInfo;
	_CurrentTrack : I_XtsTrack;
	_myStatus : MoverStatus;
	_MyCAGroup : I_CollisionGroup;
	_ForwardOnly : BOOL := TRUE;
	myControllerOid: OTCID;
	MyId: UDINT;
	MoverID : T_MaxString;
	Initialised : BOOL;
	MyTrackCount : INT;
	MyTracks : ARRAY[0..MaxTracks] OF I_XtsTrack;
	NullTrack : XtsTrack('');
	_SetForce: LREAL;
	_SetCurrent: LREAL;
	_Gap : LREAL;
	_Acceleration : LREAL;
	_Deceleration : LREAL;
	_Jerk : LREAL;
	_DistanceDrivenInMM : LREAL;
	_AvoidingCollision: BOOL;
	_Mover1 : BOOL;
	myController: Tc3_XTS_Utility.I_McXtsMoverController;
END_VAR
VAR CONSTANT
	_MaxMoverVelocity : MC_LREAL := 4000.0;
	MaxTracks : INT := 5;
	InPositionToleranceForMoveChecks : LREAL := 0.001;
END_VAR

PROPERTY PUBLIC Acceleration : MC_LREAL
GET
Acceleration := MoveBehaviour.Acceleration;
END_GET
SET
MoveBehaviour.Acceleration := Acceleration;
_Acceleration := Acceleration;
END_SET
END_PROPERTY

METHOD ActivateTrack : HRESULT
VAR_INPUT
	Track : INT;
END_VAR
IF Track = 0 THEN
	ActivateTrack := -1;
	Base_Library.Tracing.Trace.Warning(MoverID, 'ActivateTrack Fail - Null Track');
	RETURN;
END_IF
IF MoverActivateTrackBehaviour.Busy THEN
	ActivateTrack := -2;
	Base_Library.Tracing.Trace.Warning(MoverID, 'ActivateTrack Fail - Activating');
	RETURN;
END_IF

IF NOT THIS^.IsStationary THEN
	ActivateTrack := -3;
	Base_Library.Tracing.Trace.Warning(MoverID, 'ActivateTrack Fail - Moving');
	RETURN;
END_IF

IF Track > MyTrackCount THEN
	ActivateTrack := -4;
	Base_Library.Tracing.Trace.Warning(MoverID, 'ActivateTrack Fail - Track not Registered');
	RETURN;
END_IF

IF MyTracks[Track - 1].MyOTCID = 0  THEN
	ActivateTrack := -5;
	Base_Library.Tracing.Trace.Warning(MoverID, 'ActivateTrack Fail - No Track');
	RETURN;
END_IF
	
Base_Library.Tracing.Trace.Verbose(MoverID, 'ActivateTrack Request Accepted');
MoverActivateTrackBehaviour.Execute(Track := MyTracks[Track - 1]);
_ipTcIoXtsMover.SetActiveTrackObjectId(nTrackObjectId := MyTracks[Track - 1].MyOTCID);
_CurrentTrack := MyTracks[Track - 1];
END_METHOD

METHOD ActivateZeroReferenceSystem : HRESULT
IF MoverActivateTrackBehaviour.Busy THEN
	ActivateZeroReferenceSystem := -1;
	Base_Library.Tracing.Trace.Warning(MoverID, 'ActivateZeroTrack Fail - Activating');
	RETURN;
END_IF
IF NOT THIS^.IsStationary THEN
	ActivateZeroReferenceSystem := -2;
	Base_Library.Tracing.Trace.Warning(MoverID, 'ActivateZeroTrack Fail - Moving');
	RETURN;
END_IF 

Base_Library.Tracing.Trace.Verbose(MoverID, 'ActivateTrack Request Accpeted');
MoverActivateTrackBehaviour.Execute(Track := NullTrack);
_CurrentTrack := 0;
END_METHOD

PROPERTY ActualForce : LREAL
GET
ActualForce := _SetForce;
END_GET
END_PROPERTY

PROPERTY ActualPosition : LREAL
GET
ActualPosition := MyAxisRef.NcToPlc.ActPos;
END_GET
END_PROPERTY

PROPERTY ActualTrackPosition : LREAL
GET
ActualTrackPosition := _stTmsActPositions.fTrackPosition;
END_GET
END_PROPERTY

PROPERTY ActualVelocity : LREAL
GET
ActualVelocity := MyAxisRef.NcToPlc.ActVelo;
END_GET
END_PROPERTY

PROPERTY AxisRef : Reference to Axis_ref
GET
AxisRef REF= MyAxisRef;
END_GET
END_PROPERTY

METHOD PUBLIC  Cycle : HRESULT
VAR_INPUT
END_VAR
IF Initialised THEN
	TaskCollection.Cycle();
	TrackChangeTrigger(CLK := MoverActivateTrackBehaviour.Done);
	IF TrackChangeTrigger.Q THEN
		_MoverAbsMoveOptions.PositionReferenceSystem :=  MoverActivateTrackBehaviour.NewTrackId;
		_MoverAbsMoveOptions.DynamicsReferenceSystem := MoverActivateTrackBehaviour.NewTrackId;
		MoveBehaviour.Options := _MoverAbsMoveOptions;	
	END_IF
	IF _ipTcIoXtsMover <> 0 THEN
		_stTmsActPositions := _ipTcIoXtsMover.GetPositionInfo();
		_SetForce := _ipTcIoXtsMover.GetSetForce();
		_SetCurrent := _ipTcIoXtsMover.GetSetCurrent();
		_myStatus.isMover1 := _ipTcIoXtsMover.GetIsMover1();
		_myStatus.isActive := _ipTcIoXtsMover.GetIsActive();
		_myStatus.isFrozen := _ipTcIoXtsMover.GetIsFrozen();
		_myStatus.isLost := _ipTcIoXtsMover.GetIsLost();
		_myStatus.isReadyForPositioning := _ipTcIoXtsMover.GetIsReadyForPositioning();
		_myStatus.hasControllerError := _ipTcIoXtsMover.GetMoverControllerError();
		_myStatus.driveState := _ipTcIoXtsMover.GetDriveStatus();
		_DistanceDrivenInMM := _ipTcIoXtsMover.GetDistanceDriven();
	END_IF
	_AvoidingCollision := MyAxisRef.NcToPlc.StateDWord2.Flags.AvoidingCollision;
ELSE
	Cycle := -1;
END_IF
MyAxisRef.ReadStatus();
_MyNCData := MyAxisRef.NcToPlc;
_MyAxisStatus := MyAxisRef.Status;
END_METHOD

PROPERTY PUBLIC Deceleration : MC_LREAL
GET
Deceleration := MoveBehaviour.Deceleration;
END_GET
SET
MoveBehaviour.Deceleration := Deceleration;
HaltBehaviour.Deceleration := Deceleration;
_Deceleration := Deceleration;
END_SET
END_PROPERTY

METHOD PUBLIC DisableMover : HRESULT
VAR_INPUT
END_VAR
IF NOT THIS^.IsEnabled THEN
	DisableMover := -1;
	Base_Library.Tracing.Trace.Warning(MoverID, 'Disable request Fail - Disabled'); 
	RETURN;
END_IF
	
Base_Library.Tracing.Trace.Verbose(MoverID, 'Disable Request Accepted');
EnableBehaviour.Disable();
END_METHOD

METHOD PUBLIC EnableMover : HRESULT
VAR_INPUT
END_VAR
IF EnableBehaviour.Busy THEN
	EnableMover := -1;
	Base_Library.Tracing.Trace.Warning(MoverID, 'Enable Request Failed - Enabling');
	RETURN;
END_IF
IF THIS^.IsEnabled THEN
	EnableMover := -2;
	Base_Library.Tracing.Trace.Warning(MoverID, 'Enable Request Failed - Enabled');
	RETURN;
END_IF
	
Base_Library.Tracing.Trace.Verbose(MoverID, 'Enable Request Accepted');
EnableBehaviour.Enable();
END_METHOD

PROPERTY ErrorID : UDINT
GET
ErrorID := _MyAxisStatus.ErrorID;
END_GET
END_PROPERTY

//FB_Init is always available implicitly and it is used primarily for initialization.
//The return value is not evaluated. For a specific influence, you can also declare the
//methods explicitly and provide additional code there with the standard initialization
//code. You can evaluate the return value.
METHOD FB_Init: BOOL
VAR_INPUT
    bInitRetains: BOOL; // TRUE: the retain variables are initialized (reset warm / reset cold)
    bInCopyCode: BOOL;  // TRUE: the instance will be copied to the copy code afterward (online change)   
END_VAR
TaskCollection.RegisterCyclic(EnableBehaviour);
TaskCollection.RegisterCyclic(ResetBehaviour);
TaskCollection.RegisterCyclic(HaltBehaviour);
TaskCollection.RegisterCyclic(MoveBehaviour);
TaskCollection.RegisterCyclic(MoverActivateTrackBehaviour);
END_METHOD

PROPERTY PUBLIC Gap : MC_LREAL
GET
Gap := MoveBehaviour.Gap;
END_GET
SET
IF Gap >= 50.0 THEN
	MoveBehaviour.Gap := Gap;
	HaltBehaviour.Gap := Gap;
	_Gap := Gap;
ELSE
	_Gap := 100.0;
	MoveBehaviour.Gap := 100.0;
	HaltBehaviour.Gap := 100.0;
END_IF
END_SET
END_PROPERTY

METHOD GetActiveTrackLength : LREAL
VAR_INPUT
END_VAR
GetActiveTrackLength := _CurrentTrack.TrackLength;
END_METHOD

METHOD GetMoverCtrlOTCID : XtsMoverControllerOTCID
VAR_INPUT
END_VAR
GetMoverCtrlOTCID := _ipTcIoXtsMover.GetMoverControllerOid();
END_METHOD

METHOD GetMoverOTCID : OTCID
VAR_INPUT
END_VAR
//GetMoverCtrlOTCID := _ipTcIoXtsMover.P_AxisOid;
END_METHOD

METHOD PUBLIC HaltAxis : HRESULT
VAR_INPUT
END_VAR
IF HaltBehaviour.Busy THEN
	HaltAxis := -1;
	Base_Library.Tracing.Trace.Warning(MoverID, 'Halt Request Fail - Halting');
	RETURN;
END_IF
	
Base_Library.Tracing.Trace.Verbose(MoverID, 'Halt Request Accepted');
HaltBehaviour.Execute();
END_METHOD

PROPERTY HasError : BOOL
GET
HasError := _MyAxisStatus.Error;
END_GET
END_PROPERTY

PROPERTY PUBLIC IdentInGroup : IDENT_IN_GROUP_REF
GET
IdentInGroup := UDINT_TO_IDENTINGROUP(id := _MyNCData.AxisId);
END_GET
END_PROPERTY

METHOD Initialise : HRESULT
VAR_INPUT
END_VAR
VAR
	i : INT;
END_VAR
IF Initialised THEN
	Initialise := -1;
	RETURN;
END_IF
IF _ipTcIoXtsMover = 0 THEN
	Initialise := -2;
	RETURN;
END_IF
IF NOT IsDetected THEN
	Initialise := -3;
	RETURN;
END_IF
IF MyTrackCount = 0 THEN
	Initialise := -4;
	RETURN;
END_IF
myController := _ipTcIoXtsMover.MoverController;
myControllerOid := _ipTcIoXtsMover.GetMoverControllerOid();
MyId := _ipTcIoXtsMover.P_AxisId;
MoverID := CONCAT('Mover ', TO_STRING(MyId));
_Mover1 := _ipTcIoXtsMover.GetIsMover1();
_CurrentTrack := MyTracks[MoversActiveTrack - 1];
Initialised := TRUE;
END_METHOD

PROPERTY IsActive : BOOL
GET
IsActive := _myStatus.isActive;
END_GET
END_PROPERTY

PROPERTY IsAMover1 : BOOL
GET
IsAMover1 := _Mover1;
END_GET
END_PROPERTY

PROPERTY IsAvoidingCollision : BOOL
GET
isAvoidingCollision := _AvoidingCollision;
END_GET
END_PROPERTY

PROPERTY IsDetected : BOOL
GET
IsDetected := MyAxisRef.NcToPlc.AxisId <> 0;
END_GET
END_PROPERTY

PROPERTY IsEnabled : BOOL
GET
IsEnabled :=  NOT _MyAxisStatus.Disabled;
END_GET
END_PROPERTY

PROPERTY IsStationary : BOOL
GET
IsStationary := _MyAxisStatus.NotMoving;
END_GET
END_PROPERTY

PROPERTY PUBLIC Jerk : MC_LREAL
GET
Jerk := MoveBehaviour.Jerk;
END_GET
SET
MoveBehaviour.Jerk := Jerk;
HaltBehaviour.Jerk := Jerk;
_Jerk := Jerk;
END_SET
END_PROPERTY

PROPERTY PUBLIC MoversActiveTrack : INT
GET
VAR
	i : INT;
END_VAR
FOR i := 0 TO MyTrackCount - 1 DO
	IF MyTracks[i].MyOTCID =  _ipTcIoXtsMover.GetActiveTrackObjectId() THEN
		MoversActiveTrack := i + 1;
		EXIT;
	END_IF
END_FOR
END_GET
END_PROPERTY

PROPERTY PUBLIC MoverXtsIoEnvInterface : I_TcIoXtsXpuMover
GET
MoverXtsIoEnvInterface := _ipTcIoXtsMover;
END_GET
SET
_ipTcIoXtsMover := MoverXtsIoEnvInterface;
END_SET
END_PROPERTY

METHOD PUBLIC MoveTo : HRESULT
VAR_INPUT
	RequiredPosition : MC_LREAL;
	MoveVelocity : MC_LREAL;
	NonModuloMove : BOOL;
END_VAR
IF MoveBehaviour.Busy THEN
	Base_Library.Tracing.Trace.Warning(MoverID, 'Mover Called While Busy');
END_IF
IF MoveVelocity > _MaxMoverVelocity THEN
	Base_Library.Tracing.Trace.Warning(MoverID, 'Move Velo Too High');
	MoveTo := -2;
	RETURN;
END_IF
IF MoveVelocity <= 0.0 THEN
	Base_Library.Tracing.Trace.Warning(MoverID, 'Move Velo Less Than Zero');
	MoveTo := -3;
	RETURN;
END_IF
IF Gap <= 50.0 THEN
	Base_Library.Tracing.Trace.Warning(MoverID, 'Move Gasp Too Small');
	MoveTo := -4;
	RETURN;
END_IF

Base_Library.Tracing.Trace.Verbose(moverID, concat('Move Accepted to : ',TO_STRING(RequiredPosition)));

IF NonModuloMove THEN
	THIS^.MoveBehaviour.MoveTo(Position := RequiredPosition, 
									Velocity := MoveVelocity, 
									Direction := Tc3_Mc3Definitions.MC_DIRECTION.mcDirectionNonModulo, 
									Turns := 0);
	MoveTo := 1;
END_IF

IF NOT NonModuloMove AND _ForwardOnly THEN
	MoveTo := THIS^.MoveBehaviour.MoveTo(Position := RequiredPosition, 
									Velocity := MoveVelocity, 
									Direction := Tc3_Mc3Definitions.MC_DIRECTION.mcDirectionPositive, 
									Turns := 0);
	MoveTo := 2;
END_IF

IF NOT NonModuloMove AND NOT _ForwardOnly THEN
	IF RequiredPosition > MyAxisRef.NcToPlc.ModuloActPos THEN
		MoveTo := THIS^.MoveBehaviour.MoveTo(Position := RequiredPosition, 
									Velocity := MoveVelocity, 
									Direction := Tc3_Mc3Definitions.MC_DIRECTION.mcDirectionPositive, 
									Turns := 0);
		MoveTo := 3;
	ELSE
		MoveTo := THIS^.MoveBehaviour.MoveTo(Position := RequiredPosition, 
									Velocity := MoveVelocity, 
									Direction := Tc3_Mc3Definitions.MC_DIRECTION.mcDirectionNegative, 
									Turns := 0);
		MoveTo := 4;
	END_IF
END_IF
END_METHOD

PROPERTY MyCAGroup : I_CollisionGroup
GET
MyCAGroup := _MyCAGroup;
END_GET
SET
_MyCAGroup := MyCAGroup;
END_SET
END_PROPERTY

PROPERTY PositiveDirectionOnly : BOOL
GET
PositiveDirectionOnly := _ForwardOnly;
END_GET
SET
_ForwardOnly := PositiveDirectionOnly;
END_SET
END_PROPERTY

METHOD RegisterTracks : HRESULT
VAR_INPUT
	Track : I_XtsTrack;
END_VAR
VAR
	Registered : BOOL;
	i : INT;
END_VAR
IF Track = 0 THEN
	RegisterTracks := -1;
	RETURN;
END_IF
Registered := FALSE;
FOR i := 0 TO 5 DO 
	IF Track = MyTracks[i] THEN
		Registered := TRUE;
	END_IF
END_FOR
IF Registered THEN
	RegisterTracks := -2;
	RETURN;
END_IF
FOR i := 0 TO 5 DO
	IF MyTracks[i] = 0 THEN
		MyTracks[i] := Track;
		MyTrackCount := MyTrackCount + 1;
		EXIT;
	END_IF
END_FOR
END_METHOD

METHOD RegisterWithParent
VAR_INPUT
	Parent	: I_HostObjects;
END_VAR
Parent.RegisterCyclic(THIS^);
END_METHOD

METHOD PUBLIC Reset : HRESULT
VAR_INPUT
END_VAR
IF ResetBehaviour.Busy THEN
	Base_Library.Tracing.Trace.Warning(MoverID, 'Reset Request Failed - Reseting');
	Reset := -1;
	RETURN;
END_IF
 
IF NOT (_MyAxisStatus.Error OR _MyAxisStatus.NotMoving) THEN
	Base_Library.Tracing.Trace.Warning(MoverID, 'Reset Request Failed - Not Allowed');
	Reset := -2;
	RETURN;
END_IF

Base_Library.Tracing.Trace.Verbose(MoverID, 'Reset Request Accepted');
ResetBehaviour.Reset();
MoveBehaviour.Abort();
END_METHOD

METHOD SetForceCouple : HRESULT
VAR_INPUT
	XtsMoverCtrlOTCID : Tc3_XTS_Utility.XtsMoverControllerOTCID;
END_VAR
IF _ipTcIoXtsMover = 0 THEN
	SetForceCouple := - 1;
	RETURN;
END_IF

_ipTcIoXtsMover.MoverController.SetForceCouple(nForceCouple := XtsMoverCtrlOTCID);
END_METHOD

METHOD SetMoverActiveTrack : HRESULT
VAR_INPUT
	Track : INT;
END_VAR
IF Track = 0 THEN
	SetMoverActiveTrack := -1;
	RETURN;
END_IF

IF NOT THIS^.IsStationary THEN
	SetMoverActiveTrack := -3;
	RETURN;
END_IF

IF Track > MyTrackCount THEN
	SetMoverActiveTrack := -4;
	RETURN;
END_IF

IF MyTracks[Track - 1].MyOTCID = 0  THEN
	SetMoverActiveTrack := -5;
	RETURN;
END_IF
	
_ipTcIoXtsMover.SetActiveTrackObjectId(nTrackObjectId := MyTracks[Track - 1].MyOTCID);
_CurrentTrack := MyTracks[Track - 1];
END_METHOD

METHOD SetParameterSet : HRESULT
VAR_INPUT
	ParameterSet : OTCID;
END_VAR
IF ParameterSet = 0 THEN
	RETURN;
	SetParameterSet := -1;
END_IF

myController.SetDefaultParameterSet(ParameterSet);
END_METHOD

METHOD SetSimDetectionPartAndPosition : BOOL
VAR_INPUT
	Part : OTCID;
	Position : LREAL;
END_VAR
_ipTcIoXtsMover.SetSimulatedStartUpPart(Part);
_ipTcIoXtsMover.SetSimulatedStartUpPosition(Position);
END_METHOD

METHOD SwapMover : HRESULT
VAR_INPUT
    MoverToSwapWith : MoverOTCID;
END_VAR
_ipTcIoXtsMover.swapmover(nSwapMoverObjectId := MoverToSwapWith);
END_METHOD

METHOD TriggerMoverArrive : HRESULT
VAR_INPUT
END_VAR
IF _ipTcIoXtsMover = 0 THEN
	TriggerMoverArrive := - 1;
	RETURN;
END_IF
IF _myStatus.isActive THEN
	TriggerMoverArrive := - 2;
	RETURN;
END_IF

_ipTcIoXtsMover.TriggerArrive();
END_METHOD

METHOD TriggerMoverLeave : HRESULT
VAR_INPUT
END_VAR
IF _ipTcIoXtsMover = 0 THEN
	TriggerMoverLeave := -1;
	RETURN;
END_IF
IF NOT _myStatus.isActive THEN
	TriggerMoverLeave := -2;
	RETURN;
END_IF
IF NOT IsStationary THEN
	TriggerMoverLeave := -3;
	RETURN;
END_IF

_ipTcIoXtsMover.TriggerLeave();
END_METHOD

END_FUNCTION_BLOCK

// ---- Tasks/MoveToPositionTask.TcPOU
FUNCTION_BLOCK MoveToPositionTask IMPLEMENTS I_Task, I_Cyclic, I_Object, I_Abortable
VAR
	moveAbs	: MC_MoveAbsoluteCA;
	_Axis : REFERENCE TO AXIS_REF;
	_stOptions : ST_MoveAbsoluteCAOptions;
	_Done: BOOL;
	_Error: BOOL;
	_ErrorId: UDINT;
END_VAR

{analysis -2}

METHOD Abort : HRESULT
moveAbs.Execute := FALSE;
moveAbs.Position := moveAbs.Velocity := 0;
END_METHOD

PROPERTY PUBLIC Acceleration : mc_lreal
GET
Acceleration := moveAbs.Acceleration;
END_GET
SET
IF Acceleration > 0.0 THEN
	moveAbs.Acceleration := Acceleration;
END_IF
END_SET
END_PROPERTY

PROPERTY AxisRef : reference to Axis_ref
GET
AxisRef	REF= _Axis;
END_GET
SET
_Axis REF= AxisRef;
END_SET
END_PROPERTY

PROPERTY Busy : BOOL
GET
Busy := moveAbs.Busy;
END_GET
END_PROPERTY

METHOD Cycle : HRESULT
VAR_INPUT
END_VAR
IF NOT __ISVALIDREF(_Axis) THEN
	Cycle := -1;
	RETURN;
END_IF
_Done := moveAbs.Done OR _Done;
_Error := moveAbs.Error OR _Error;
IF moveAbs.ErrorId <> 0 THEN
	_ErrorId := moveAbs.ErrorId;
END_IF
moveAbs(Axis := _Axis, Options := _stOptions);
moveAbs.Execute := false;
END_METHOD

PROPERTY PUBLIC Deceleration : mc_lreal
GET
Deceleration := moveAbs.Deceleration;
END_GET
SET
IF Deceleration > 0.0 THEN
	moveAbs.Deceleration := Deceleration;
END_IF
END_SET
END_PROPERTY

PROPERTY Done : BOOL
GET
Done := _Done;
END_GET
END_PROPERTY

PROPERTY Error : BOOL
GET
Error := _Error;
END_GET
END_PROPERTY

PROPERTY PUBLIC Gap : mc_lreal
GET
Gap := moveAbs.Gap;
END_GET
SET
IF Gap > 50.0 THEN
	moveAbs.Gap := Gap;
END_IF
END_SET
END_PROPERTY

PROPERTY PUBLIC Jerk : mc_lreal
GET
Jerk := moveAbs.Jerk;
END_GET
SET
IF Jerk > 0.0 THEN
	moveAbs.Jerk := Jerk;
END_IF
END_SET
END_PROPERTY

METHOD MoveTo : HRESULT
VAR_INPUT
	Position : MC_LREAL;
	Velocity : MC_LREAL;
	Direction: Tc3_Mc3Definitions.MC_DIRECTION;
	Turns: UDINT;
END_VAR
IF moveAbs.Execute THEN
	MoveTo := -1;
	RETURN;
END_IF
	
IF NOT __ISVALIDREF(_Axis) THEN
	MoveTo := -2;
	RETURN;
END_IF

IF Velocity <= 0.0 THEN
	MoveTo := -3;
	RETURN;
END_IF

moveAbs.Position := Position;
moveAbs.Velocity := Velocity;
moveAbs.Direction := Direction;
moveAbs.Options.AdditionalTurns := Turns;
moveAbs.Execute := TRUE;
_Error := FALSE;
_ErrorId := 0;
_Done := FALSE;
END_METHOD

PROPERTY PUBLIC Options : ST_MoveAbsoluteCAOptions
GET
Options := _stOptions;
END_GET
SET
_stOptions := Options;
END_SET
END_PROPERTY

METHOD RegisterWithParent
VAR_INPUT
	Parent	: Base_Library.I_HostObjects;
END_VAR
Parent.RegisterCyclic(THIS^);
Parent.RegisterAbortable(THIS^);
Parent.RegisterTask(THIS^);
END_METHOD

END_FUNCTION_BLOCK

// ---- Tasks/HaltMoverTask.TcPOU
FUNCTION_BLOCK HaltMoverTask  IMPLEMENTS I_Task, I_Object, I_Cyclic, I_Abortable
VAR
	haltMoverCA : Tc3_McCollisionAvoidance.MC_HaltCA;
	_Axis : REFERENCE TO Tc2_MC2.AXIS_REF;
	_Error: BOOL;
	_ErrorID: UDINT;
	_Done: BOOL;
END_VAR

{analysis -2}

METHOD Abort : Hresult
haltMoverCA.Execute := FALSE;
END_METHOD

PROPERTY AxisRef : reference to Axis_ref
GET
AxisRef	REF= _Axis;
END_GET
SET
_Axis REF= AxisRef;
END_SET
END_PROPERTY

PROPERTY Busy : BOOL
GET
Busy := haltMoverCA.Busy;
END_GET
END_PROPERTY

METHOD Cycle : HRESULT
VAR_INPUT
END_VAR
IF NOT __ISVALIDREF(_Axis) THEN
	Cycle := -1;
	RETURN;
END_IF

haltMoverCA(Axis := _Axis);
_Done := haltMoverCA.Done OR _Done;
_Error := haltMoverCA.Error OR _Error;
IF haltMoverCA.ErrorId <> 0 THEN
	_ErrorID := haltMoverCA.ErrorId;
END_IF
haltMoverCA.Execute := false;
END_METHOD

PROPERTY Deceleration : MC_LREAL
GET
Deceleration := haltMoverCA.Deceleration;
END_GET
SET
IF Deceleration > 0.0 THEN
	haltMoverCA.Deceleration := Deceleration;
END_IF
END_SET
END_PROPERTY

PROPERTY Done : BOOL
GET
Done := _Done;
END_GET
END_PROPERTY

PROPERTY Error : BOOL
GET
Error := _Error;
END_GET
END_PROPERTY

METHOD Execute : HRESULT
VAR_INPUT
END_VAR
IF haltMoverCA.Execute THEN
	Execute := -1;
	RETURN;
END_IF

IF NOT __ISVALIDREF(_axis) THEN
	Execute	 := -1;
	RETURN;
END_IF

haltMoverCA.Execute := TRUE;
_Error := FALSE;
_ErrorId := 0;
_Done := FALSE;
END_METHOD

PROPERTY Gap : MC_LREAL
GET
Gap := haltMoverCA.Gap;
END_GET
SET
IF Gap > 50.0 THEN
	haltMoverCA.Gap := Gap;
END_IF
END_SET
END_PROPERTY

PROPERTY Jerk : MC_LREAL
GET
Jerk := haltMoverCA.Jerk;
END_GET
SET
IF Jerk > 0.0 THEN
	haltMoverCA.Jerk := Jerk;
END_IF
END_SET
END_PROPERTY

METHOD RegisterWithParent
VAR_INPUT
	Parent	: Base_Library.I_HostObjects;
END_VAR
Parent.RegisterCyclic(THIS^);
Parent.RegisterAbortable(THIS^);
Parent.RegisterTask(THIS^);
END_METHOD

END_FUNCTION_BLOCK

// ---- Tasks/ActivateTrackTask.TcPOU
FUNCTION_BLOCK ActivateTrackTask IMPLEMENTS I_Task, I_Cyclic, I_Object, I_Abortable
VAR
	mcActivateTrack : Tc3_McCollisionAvoidance.MC_ActivateTrack;
	_Axis : REFERENCE TO Tc2_MC2.AXIS_REF;
	_newTrackId : OTCID;
	_Done : BOOL;
	_Error : BOOL;
	_ErrorId : UDINT;
END_VAR

{analysis -2}

METHOD Abort : HRESULT
mcActivateTrack.Execute := FALSE;
END_METHOD

PROPERTY AxisRef : reference to Axis_ref
GET
AxisRef	REF= _Axis;
END_GET
SET
_Axis REF= AxisRef;
END_SET
END_PROPERTY

PROPERTY Busy : BOOL
GET
Busy := mcActivateTrack.Busy;
END_GET
END_PROPERTY

METHOD Cycle : HRESULT
VAR_INPUT
END_VAR
IF NOT __ISVALIDREF(_Axis) THEN
	Cycle := -1;
	RETURN;
END_IF
_Done := mcActivateTrack.Done OR _Done;
_Error := mcActivateTrack.Error OR _Error;
IF mcActivateTrack.ErrorId <> 0 THEN
	_ErrorId := mcActivateTrack.ErrorId;
END_IF
_newTrackId := mcActivateTrack.TrackId;
mcActivateTrack(Axis := _Axis);
mcActivateTrack.Execute := FALSE;
END_METHOD

PROPERTY Done : BOOL
GET
Done := _Done;
END_GET
END_PROPERTY

PROPERTY Error : BOOL
GET
Error := _Error;
END_GET
END_PROPERTY

METHOD PUBLIC Execute : HRESULT
VAR_INPUT
	Track : I_XtsTrack;
END_VAR
IF mcActivateTrack.Execute THEN
	Execute := -1;
	RETURN;
END_IF

IF Track = 0 THEN
	Execute := -2;
	RETURN;
END_IF

IF NOT __ISVALIDREF(_Axis) THEN
	Execute := - 3;
	RETURN;
END_IF;

IF _Axis.Status.Disabled THEN
	Execute := -4;
	RETURN;
END_IF

IF _Axis.NcToPlc.SetVelo <> 0.0 THEN
	Execute := -5;
	RETURN;
END_IF

mcActivateTrack.Execute := TRUE;
mcActivateTrack.TrackId := Track.MyOTCID;
_Error := FALSE;
_ErrorId := 0;
_Done := FALSE;
END_METHOD

PROPERTY PUBLIC NewTrackId : OTCID
GET
NewTrackId := _newTrackId;
END_GET
END_PROPERTY

METHOD RegisterWithParent
VAR_INPUT
	Parent	: Base_Library.I_HostObjects;
END_VAR
Parent.RegisterCyclic(THIS^);
Parent.RegisterAbortable(THIS^);
Parent.RegisterTask(THIS^);
END_METHOD

END_FUNCTION_BLOCK

// ---- Hardware/XtsTrack.TcPOU
FUNCTION_BLOCK XtsTrack EXTENDS CyclicBase IMPLEMENTS I_XtsTrack, I_Initialisable
VAR
	_MyInterface : I_TcIoXtsXpuTrack;
	XtsIoEnvInitialiseState : INT;
	MyPartCount : UDINT;
	Parts : REFERENCE TO ARRAY[1..TcIoXtsEnvironmentParameterList.MaxPartsPerTrack] OF ST_PartInfoItems;
	_TrackLength: LREAL;
	_TrackIsClosed: BOOL;
	_OTCID : OTCID;
	_IsTrackIncludedForDetection : BOOL;
	_NumberOfPartsInTrack : INT;
	_TrackPolarity: Tc3_XTS_Utility.Polarity;
	_IsInitialised : BOOL;
END_VAR

METHOD PUBLIC  Cycle : HRESULT
VAR_INPUT
END_VAR
IF _MyInterface = 0 THEN
	Cycle := -1;
	RETURN;
END_IF

_IsTrackIncludedForDetection := _MyInterface.GetIsIncludedInDetection();
END_METHOD

METHOD Initialise : HRESULT
VAR_INPUT
END_VAR
Initialise := -1;
CASE XtsIoEnvInitialiseState OF
	0:
		IF _MyInterface <> 0 THEN
			XtsIoEnvInitialiseState := 1;
		ELSE
			XtsIoEnvInitialiseState := 999;
		END_IF
	1:
		MyPartCount := _MyInterface.GetPartCount();
		XtsIoEnvInitialiseState := 2;
	2:
		XtsIoEnvInitialiseState := 3;
		Parts REF= _MyInterface.GetPartInfoItems();
		
	3:
		IF _MyInterface.P_IsInitialized THEN
			_TrackLength := _MyInterface.GetLength();
			_TrackIsClosed := _MyInterface.GetIsClosed();
			_TrackPolarity := _MyInterface.GetPolarity();
			_NumberOfPartsInTrack := TO_INT(_MyInterface.GetPartCount());
			XtsIoEnvInitialiseState := 4;
		END_IF
	4:
		Initialise := 0;
		_IsInitialised := TRUE;
END_CASE
END_METHOD

PROPERTY Initialised : BOOL
GET
Initialised := _IsInitialised;
END_GET
END_PROPERTY

PROPERTY IsTrackSetForDetection : BOOL
GET
IsTrackSetForDetection := _IsTrackIncludedForDetection;
END_GET
END_PROPERTY

PROPERTY MyOTCID : OTCID
GET
MyOTCID := _OTCID;
END_GET
SET
_OTCID := MyOTCID;
END_SET
END_PROPERTY

PROPERTY MyXtsIoEnvInterface : I_TcIoXtsXpuTrack
GET
MyXtsIoEnvInterface := _MyInterface;
END_GET
SET
_MyInterface := MyXtsIoEnvInterface;
END_SET
END_PROPERTY

PROPERTY NumberOfPartsInTrack : INT
GET
NumberOfPartsInTrack := _NumberOfPartsInTrack;
END_GET
END_PROPERTY

METHOD RemoveFromDetection : BOOL
VAR_INPUT
END_VAR
RemoveFromDetection := _MyInterface.SetIsIncludedInDetection(False);
END_METHOD

METHOD SetForDetection : BOOL
VAR_INPUT
END_VAR
SetForDetection := _MyInterface.SetIsIncludedInDetection(TRUE);
END_METHOD

PROPERTY TrackLength : MC_Lreal
GET
TrackLength := _MyInterface.GetLength();
END_GET
END_PROPERTY

END_FUNCTION_BLOCK

// ---- Tasks/AddMoverToGroupTask.TcPOU
FUNCTION_BLOCK AddMoverToGroupTask IMPLEMENTS I_Task
VAR_INPUT
END_VAR
VAR_OUTPUT
END_VAR
VAR
	AddtoGrp			: MC_AddAxisToGroup;
	_CaGroup			: I_CollisionGroup;
	_Axis				: REFERENCE TO AXIS_REF;
	_Done 				: BOOL;
	_Error				: BOOL;
	_ErrorID			: UDINT;
END_VAR

{analysis -2}

METHOD Abort : BOOL
AddtoGrp.Execute := FALSE;
Abort := true;
END_METHOD

METHOD AddMover : hresult
VAR_INPUT
	MoverToAdd : I_XtsMover;
END_VAR
IF MoverToAdd = 0 THEN
	AddMover := -1;
	RETURN;
END_IF

IF AddtoGrp.Execute THEN
	AddMover := -2;
	RETURN;
END_IF
	
AddtoGrp.Execute := TRUE;
AddtoGrp.IdentInGroup := MoverToAdd.IdentInGroup;
_Axis REF= MoverToAdd.AxisRef;
_Error := FALSE;
_ErrorId := 0;
_Done := FALSE;
END_METHOD

PROPERTY Busy : BOOL
GET
Busy := AddtoGrp.Busy;
END_GET
END_PROPERTY

METHOD Cycle : HRESULT
VAR_INPUT
END_VAR
IF _CaGroup = 0 OR NOT __ISVALIDREF(_Axis) THEN
	Cycle := -1;
	RETURN;
END_IF
_Done := AddtoGrp.Done OR _Done;
_Error := AddtoGrp.Error OR _Error;
IF AddtoGrp.ErrorId <> 0 THEN
	_ErrorId := AddtoGrp.ErrorId;
END_IF
AddtoGrp(AxesGroup := _CaGroup.GroupRef,
			Axis := _Axis);
AddtoGrp.Execute := FALSE;
END_METHOD

PROPERTY Done : BOOL
GET
Done := _Done;
END_GET
END_PROPERTY

PROPERTY Error : BOOL
GET
Error := _Error;
END_GET
END_PROPERTY

PROPERTY MyCollisionGroup : I_CollisionGroup
GET
MyCollisionGroup := _caGroup;
END_GET
SET
IF MyCollisionGroup <> 0 THEN
	_caGroup := MyCollisionGroup;
END_IF
END_SET
END_PROPERTY

END_FUNCTION_BLOCK

// ---- Tasks/DisableGroup.TcPOU
FUNCTION_BLOCK DisableGroup  IMPLEMENTS I_Task
VAR
	groupDisable		: MC_GroupDisable;
	_caGroup			: I_CollisionGroup;
	_Done 				: BOOL;
	_Error				: BOOL;
	_ErrorID			: UDINT;
END_VAR

{analysis -2}

METHOD Abort : BOOL
groupDisable.Execute := FALSE;
Abort := true;
END_METHOD

PROPERTY Busy : BOOL
GET
Busy := groupDisable.Busy;
END_GET
END_PROPERTY

METHOD Cycle : HRESULT
VAR_INPUT
END_VAR
IF _caGroup = 0 THEN
	cycle := -1;
	RETURN;
END_IF
_Done := groupDisable.Done OR _Done;
_Error := groupDisable.Error OR _Error;
IF groupDisable.ErrorId <> 0 THEN
	_ErrorId := groupDisable.ErrorId;
END_IF
groupDisable(AxesGroup := _caGroup.GroupRef);
groupDisable.Execute := false;
END_METHOD

PROPERTY Done : BOOL
GET
Done := _Done;
END_GET
END_PROPERTY

PROPERTY Error : BOOL
GET
Error := _Error;
END_GET
END_PROPERTY

METHOD Execute : hresult
IF groupDisable.Execute THEN
	Execute := -1;
	RETURN;
END_IF

IF _caGroup = 0 THEN
	Execute := -2;
	RETURN;
END_IF
groupDisable.Execute := TRUE;
END_METHOD

PROPERTY MyCollisionGroup : I_CollisionGroup
GET
MyCollisionGroup := _caGroup;
END_GET
SET
IF MyCollisionGroup <> 0 THEN
	_caGroup := MyCollisionGroup;
END_IF
END_SET
END_PROPERTY

END_FUNCTION_BLOCK

// ---- Tasks/EnableGroup.TcPOU
FUNCTION_BLOCK EnableGroup  IMPLEMENTS I_Task
VAR
	groupEnable			: MC_GroupEnable;
	_caGroup			: I_CollisionGroup;
	_Done 				: BOOL;
	_Error				: BOOL;
	_ErrorID			: UDINT;
END_VAR

{analysis -2}

METHOD Abort : BOOL
groupEnable.Execute := FALSE;
Abort := TRUE;
END_METHOD

PROPERTY Busy : BOOL
GET
Busy := groupEnable.Busy;
END_GET
END_PROPERTY

METHOD Cycle : HRESULT
VAR_INPUT
END_VAR
IF _caGroup = 0 THEN
	cycle := -1;
	RETURN;
END_IF
_Done := groupEnable.Done OR _Done;
_Error := groupEnable.Error OR _Error;
IF groupEnable.ErrorId <> 0 THEN
	_ErrorId := groupEnable.ErrorId;
END_IF
groupEnable(AxesGroup := _caGroup.GroupRef);
groupEnable.Execute := FALSE;
END_METHOD

PROPERTY Done : BOOL
GET
Done := _Done;
END_GET
END_PROPERTY

PROPERTY Error : BOOL
GET
Error := _Error;
END_GET
END_PROPERTY

METHOD Execute : HRESULT
IF groupEnable.Execute THEN
	Execute := -1;
	RETURN;
END_IF

IF _caGroup = 0 THEN
	Execute := -2;
	RETURN;
END_IF

groupEnable.Execute := TRUE;
END_METHOD

PROPERTY MyCollisionGroup : I_CollisionGroup
GET
MyCollisionGroup := _caGroup;
END_GET
SET
IF MyCollisionGroup <> 0 THEN
	_caGroup := MyCollisionGroup;
END_IF
END_SET
END_PROPERTY

END_FUNCTION_BLOCK

// ---- Tasks/GearCATask.TcPOU
FUNCTION_BLOCK PUBLIC GearCATask  IMPLEMENTS I_Task, I_Cyclic, I_Abortable, I_Object
VAR
	GearInPosCA : Tc3_McCollisionAvoidance.MC_GearInPosCA;
	_syncStrategy : Tc3_Mc3Definitions.MC_SYNC_STRATEGY := Tc3_Mc3Definitions.MC_SYNC_STRATEGY.mcSyncStrategyEarly;
	_SlaveAxis : I_XtsMover;
	_MasterAxis : I_XtsMover;
	_Error : BOOL;
	_ErrorID: UDINT;
	_Options: Tc3_McCollisionAvoidance.ST_GearInPosCAOptions;
END_VAR

{analysis -2}

METHOD Abort : HRESULT
GearInPosCA.Execute := FALSE;
END_METHOD

PROPERTY Busy : BOOL
GET
Busy := GearInPosCA.Busy;
END_GET
END_PROPERTY

METHOD ClearAxes : HRESULT
VAR_INPUT
END_VAR
_MasterAxis := 0;
_SlaveAxis := 0;
END_METHOD

METHOD Cycle : HRESULT
VAR_INPUT
END_VAR
IF _MasterAxis = 0 OR _SlaveAxis = 0 THEN
	Cycle := -1;
	RETURN;
END_IF
_Error := GearInPosCA.Error OR _Error;
IF  GearInPosCA.ErrorId <> 0 THEN
	_ErrorID := GearInPosCA.ErrorId;	
END_IF
GearInPosCA(Master := _MasterAxis.AxisRef, 
			Slave := _SlaveAxis.AxisRef, 
			SyncStrategy := _syncStrategy, 
			Velocity := 2000.0, 
			RatioNumerator := 1, 
			Options := _Options);
GearInPosCA.Execute := FALSE;
END_METHOD

PROPERTY Done : BOOL
GET
Done := not GearInPosCA.Busy;
END_GET
END_PROPERTY

PROPERTY Error : BOOL
GET
Error := _Error;
END_GET
END_PROPERTY

PROPERTY Gap : lreal
GET
Gap := GearInPosCA.Gap;
END_GET
SET
GearInPosCA.Gap := Gap;
END_SET
END_PROPERTY

METHOD PUBLIC GearIn : HRESULT
VAR_INPUT
	MasterPosition : MC_LREAL;
	SlavePosition : MC_LREAL;
END_VAR
IF GearInPosCA.Execute THEN
	GearIn := -1;
	RETURN;
END_IF

IF _SlaveAxis = 0 THEN
	GearIn := -2;
	RETURN;
END_IF

IF _MasterAxis = 0 THEN
	GearIn := -3;
	RETURN;
END_IF

GearInPosCA.MasterSyncPosition := MasterPosition;
GearInPosCA.SlaveSyncPosition := SlavePosition;
GearInPosCA.Execute := TRUE;
_Error := FALSE;
_ErrorID := 0;
END_METHOD

PROPERTY InGear : BOOL
GET
InGear := GearInPosCA.InSync;
END_GET
END_PROPERTY

PROPERTY MasterAxis : I_XtsMover
GET
MasterAxis := _MasterAxis;
END_GET
SET
IF (MasterAxis <> 0) AND (MasterAxis <> _SlaveAxis)  THEN
	_MasterAxis := MasterAxis;
END_IF
END_SET
END_PROPERTY

PROPERTY Options : ST_GearInPosCAOptions
GET
Options := _Options;
END_GET
SET
_Options := Options;
END_SET
END_PROPERTY

METHOD RegisterWithParent
VAR_INPUT
	Parent	: Base_Library.I_HostObjects;
END_VAR
Parent.RegisterCyclic(THIS^);
Parent.RegisterAbortable(THIS^);
Parent.RegisterTask(THIS^);
END_METHOD

PROPERTY SlaveAxis : I_XtsMover
GET
SlaveAxis := _SlaveAxis;
END_GET
SET
IF (SlaveAxis <> 0) AND (SlaveAxis <> _MasterAxis) THEN
	_SlaveAxis := SlaveAxis;
END_IF
END_SET
END_PROPERTY

PROPERTY PUBLIC SyncStrategy : mc_sync_strategy
GET
SyncStrategy := _syncStrategy;
END_GET
SET
_syncStrategy := SyncStrategy;
END_SET
END_PROPERTY

END_FUNCTION_BLOCK

// ---- Tasks/RemoveAllMoverFromGroup.TcPOU
FUNCTION_BLOCK RemoveAllMoverFromGroup  IMPLEMENTS I_Task
VAR
	RemoveAllFromGrp			: MC_UngroupAllAxes;
	_caGroup			: I_CollisionGroup;
	_Done 				: BOOL;
	_Error				: BOOL;
	_ErrorID			: UDINT;
END_VAR

{analysis -2}

METHOD Abort : BOOL
RemoveAllFromGrp.Execute := FALSE;
Abort := true;
END_METHOD

PROPERTY Busy : BOOL
GET
Busy := RemoveAllFromGrp.Busy;
END_GET
END_PROPERTY

METHOD Cycle : HRESULT
VAR_INPUT
END_VAR
IF _caGroup = 0 THEN
	Cycle := -1;
	RETURN;
END_IF

_Done := RemoveAllFromGrp.Done OR _Done;
_Error := RemoveAllFromGrp.Error OR _Error;
IF RemoveAllFromGrp.ErrorId <> 0 THEN
	_ErrorId := RemoveAllFromGrp.ErrorId;
END_IF
RemoveAllFromGrp(AxesGroup := _caGroup.GroupRef);
RemoveAllFromGrp.Execute := FALSE;
END_METHOD

PROPERTY Done : BOOL
GET
Done := _Done;
END_GET
END_PROPERTY

PROPERTY Error : BOOL
GET
Error := _Error;
END_GET
END_PROPERTY

PROPERTY MyCollisionGroup : I_CollisionGroup
GET
MyCollisionGroup := _caGroup;
END_GET
SET
IF MyCollisionGroup <> 0 THEN
	_caGroup := MyCollisionGroup;
END_IF
END_SET
END_PROPERTY

METHOD RemoveAllMover : HRESULT
IF RemoveAllFromGrp.Execute THEN
	RemoveAllMover := -1;
	RETURN;
END_IF
	
IF _caGroup = 0 THEN
	RemoveAllMover := -2;
	RETURN;
END_IF

RemoveAllFromGrp.Execute := TRUE;
END_METHOD

END_FUNCTION_BLOCK

// ---- Tasks/RemoveMoverFromGroup.TcPOU
FUNCTION_BLOCK RemoveMoverFromGroup  IMPLEMENTS I_Task
VAR
	mcRemoveAxisFromGroup : MC_RemoveAxisFromGroup;
	_caGroup : I_CollisionGroup;
	_Leave: BOOL;
	State: INT;
	_Done: BOOL;
	_Error: BOOL;
	_Busy: BOOL;
	_ErrorId : UDINT;
END_VAR

METHOD Abort : BOOL
mcRemoveAxisFromGroup.Execute := FALSE;
_Leave := FALSE;
Abort := true;
State := 0;
END_METHOD

PROPERTY Busy : BOOL
GET
Busy := _Busy;
END_GET
END_PROPERTY

METHOD Cycle : HRESULT
VAR_INPUT
END_VAR
IF _caGroup = 0 THEN
	Cycle := -1;
	RETURN;
END_IF

_Done := mcRemoveAxisFromGroup.Done OR _Done;
_Error := mcRemoveAxisFromGroup.Error OR _Error;
IF mcRemoveAxisFromGroup.ErrorId <> 0 THEN
	_ErrorId := mcRemoveAxisFromGroup.ErrorId;
END_IF

mcRemoveAxisFromGroup(AxesGroup := _caGroup.GroupRef);
mcRemoveAxisFromGroup.Execute := FALSE;
END_METHOD

PROPERTY Done : BOOL
GET
Done := _Done;
END_GET
END_PROPERTY

PROPERTY Error : BOOL
GET
Error := _Error;
END_GET
END_PROPERTY

METHOD Execute : HRESULT
VAR_INPUT
	AxisID : IDENT_IN_GROUP_REF;
END_VAR
IF mcRemoveAxisFromGroup.Execute THEN
	Execute := -1;
	RETURN;
END_IF

IF _caGroup = 0 THEN
	Execute := -2;
	RETURN;
END_IF

mcRemoveAxisFromGroup.Execute := TRUE;
mcRemoveAxisFromGroup.IdentInGroup := AxisID;
END_METHOD

PROPERTY MyCollisionGroup : I_CollisionGroup
GET
MyCollisionGroup := _caGroup;
END_GET
SET
IF MyCollisionGroup <> 0 THEN
	_caGroup := MyCollisionGroup;
END_IF
END_SET
END_PROPERTY

END_FUNCTION_BLOCK

// ---- Tasks/ResetGroup.TcPOU
FUNCTION_BLOCK ResetGroup  IMPLEMENTS I_Task
VAR
	groupReset			: MC_GroupReset;
	_caGroup			: I_CollisionGroup;
	_Done 				: BOOL;
	_Error				: BOOL;
	_ErrorID			: UDINT;
END_VAR

{analysis -2}

METHOD Abort : BOOL
groupReset.Execute := FALSE;
Abort := TRUE;
END_METHOD

PROPERTY Busy : BOOL
GET
Busy := groupReset.Busy;
END_GET
END_PROPERTY

METHOD Cycle : HRESULT
VAR_INPUT
END_VAR
IF _caGroup = 0 THEN
	cycle := -1;
	RETURN;
END_IF
_Done := groupReset.Done OR _Done;
_Error := groupReset.Error OR _Error;
IF groupReset.ErrorId <> 0 THEN
	_ErrorId := groupReset.ErrorId;
END_IF
groupReset(AxesGroup := _caGroup.GroupRef);
groupReset.Execute := FALSE;
END_METHOD

PROPERTY Done : BOOL
GET
Done := _Done;
END_GET
END_PROPERTY

PROPERTY Error : BOOL
GET
Error := _Error;
END_GET
END_PROPERTY

METHOD Execute : HRESULT
IF groupReset.Execute THEN
	Execute := -1;
	RETURN;
END_IF

IF _caGroup = 0 THEN
	Execute := -2;
	RETURN;
END_IF

groupReset.Execute := TRUE;
END_METHOD

PROPERTY MyCollisionGroup : I_CollisionGroup
GET
MyCollisionGroup := _caGroup;
END_GET
SET
IF MyCollisionGroup <> 0 THEN
	_caGroup := MyCollisionGroup;
END_IF
END_SET
END_PROPERTY

END_FUNCTION_BLOCK

// ---- Tasks/StopMoverGroup.TcPOU
FUNCTION_BLOCK StopMoverGroup  IMPLEMENTS I_Task
VAR
	groupStop			: MC_GroupStop;
	_caGroup			: I_CollisionGroup;
	_Done 				: BOOL;
	_Error				: BOOL;
	_ErrorID			: UDINT;
END_VAR

{analysis -2}

METHOD Abort : BOOL
groupStop.Execute := FALSE;
Abort := TRUE;
END_METHOD

PROPERTY Busy : BOOL
GET
Busy := groupStop.Busy;
END_GET
END_PROPERTY

METHOD Cycle : HRESULT
VAR_INPUT
END_VAR
IF _caGroup = 0 THEN
	cycle := -1;
	RETURN;
END_IF
_Done := groupStop.Done OR _Done;
_Error := groupStop.Error OR _Error;
IF groupStop.ErrorId <> 0 THEN
	_ErrorId := groupStop.ErrorId;
END_IF
groupStop(AxesGroup := _caGroup.GroupRef);
groupStop.Execute := FALSE;
END_METHOD

PROPERTY PUBLIC Deceleration : MC_LREAL
GET
Deceleration := groupStop.Deceleration;
END_GET
SET
IF Deceleration > 0.0 THEN
	groupStop.Deceleration := Deceleration;
END_IF
END_SET
END_PROPERTY

PROPERTY Done : BOOL
GET
Done := _Done;
END_GET
END_PROPERTY

PROPERTY Error : BOOL
GET
Error := _Error;
END_GET
END_PROPERTY

METHOD Execute : HRESULT
IF groupStop.Execute THEN
	Execute := -1;
	RETURN;
END_IF

IF _caGroup = 0 THEN
	Execute := -2;
	RETURN;
END_IF

groupStop.Execute := TRUE;
END_METHOD

PROPERTY PUBLIC Jerk : MC_LREAL
GET
Jerk := groupStop.Jerk;
END_GET
SET
IF Jerk > 0.0 THEN
	groupStop.Jerk := Jerk;
END_IF
END_SET
END_PROPERTY

PROPERTY MyCollisionGroup : I_CollisionGroup
GET
MyCollisionGroup := _caGroup;
END_GET
SET
IF MyCollisionGroup <> 0 THEN
	_caGroup := MyCollisionGroup;
END_IF
END_SET
END_PROPERTY

END_FUNCTION_BLOCK

// ---- XPU/XtsIoEnvVar.TcPOU
FUNCTION_BLOCK XtsIoEnvVar IMPLEMENTS I_XtsIoEnvVar, I_Object, I_Initialisable
VAR
	XtsIoEnvironment : Tc3_XTS_Utility.FB_TcIoXtsEnvironment;
	stXtsEnvironmentConfiguration	: ST_XtsEnvironmentConfiguration;
	_Initialised : BOOL;
END_VAR

METHOD FB_init : BOOL
VAR_INPUT
	bInitRetains : BOOL; // if TRUE, the retain variables are initialized (warm start / cold start)
	bInCopyCode : BOOL;  // if TRUE, the instance afterwards gets moved into the copy code (online change)
END_VAR
stXtsEnvironmentConfiguration.bEnableInitCaGroup := TRUE;
XtsIoEnvironment.P_XtsEnvironmentConfiguration := stXtsEnvironmentConfiguration;
END_METHOD

METHOD GetCaGroupInterface : I_Mc2CaGroup
VAR_INPUT
	CAGroupNumber : INT;
END_VAR
IF NOT Initialised THEN
	RETURN;
END_IF

GetCaGroupInterface := XtsIoEnvironment.Mc2CaGroup(TO_UINT(CAGroupNumber));
END_METHOD

METHOD GetXPUInterface : I_TcIoXtsProcessingUnit
VAR_INPUT
	MyXts : INT;
END_VAR
IF NOT Initialised THEN
	RETURN;
END_IF

GetXPUInterface := XtsIoEnvironment.XpuTcIo(TO_UINT(MyXts));
END_METHOD

METHOD PUBLIC Initialise : HRESULT
VAR_INPUT
END_VAR
IF XtsIoEnvironment.Init(TRUE) THEN
	XtsIoEnvironment.Init(FALSE);
	_Initialised := TRUE;
ELSE
	Initialise := -1;
END_IF
END_METHOD

PROPERTY Initialised : BOOL
GET
Initialised := _Initialised;
END_GET
END_PROPERTY

METHOD RegisterWithParent
VAR_INPUT
	Parent	: I_HostObjects;
END_VAR
Parent.RegisterInitialisable(THIS^);
END_METHOD

END_FUNCTION_BLOCK

// ---- Collision Group/CollisionGroup.TcPOU
FUNCTION_BLOCK CollisionGroup IMPLEMENTS I_Cyclic, I_CollisionGroup, I_Resettable, I_Object
VAR
	stGroupInformation : CAGroupInfo;
	_caGroup : Tc3_McCoordinatedMotion.AXES_GROUP_REF;
	_ICaGroup : I_Mc2CaGroup;
	ReadGroupStatus : Tc3_McCoordinatedMotion.MC_GroupReadStatus;
	ReadErrorCode : Tc3_McCoordinatedMotion.MC_GroupReadError;
	resetCAGroup : ResetGroup := (MyCollisionGroup := THIS^);
	enableCAGroup : EnableGroup := (MyCollisionGroup := THIS^);
	disableCAGroup : DisableGroup := (MyCollisionGroup := THIS^);
	addMover : AddMoverToGroupTask := (MyCollisionGroup := THIS^);
	removeAllAxes : RemoveAllMoverFromGroup := (MyCollisionGroup := THIS^);
	grpStop : StopMoverGroup := (MyCollisionGroup := THIS^);
	removeMover : RemoveMoverFromGroup := (MyCollisionGroup := THIS^);
	_MyName: STRING;
	GroupMovers : ARRAY[0..MaxMovers] OF I_XtsMover;
	RegisteredMovers : INT;
	GroupErrorCode: UDINT;
END_VAR
VAR CONSTANT
	MaxMovers : INT := 49;
END_VAR

{analysis -2}

METHOD AddMoverToThisGroup : HRESULT
VAR_INPUT
	MoverToAdd : I_XtsMover;
END_VAR
VAR
	i : INT;
	Registered : BOOL;
END_VAR
IF MoverToAdd = 0 THEN
	Base_Library.Tracing.Trace.Warning(_MyName, 'Register Mover Fail - null ptr');
	AddMoverToThisGroup := -1;
	RETURN;
END_IF
FOR i := 0 TO MaxMovers DO
	IF GroupMovers[i] = MoverToAdd THEN
		registered := TRUE;
	END_IF
END_FOR
IF registered THEN
	Base_Library.Tracing.Trace.Warning(_MyName, 'Register Mover Fail - registered');
	AddMoverToThisGroup := -2;
	RETURN;
END_IF
IF addMover.Busy THEN
	Base_Library.Tracing.Trace.Warning(_MyName, 'Register Mover Fail - busy');
	AddMoverToThisGroup := -3;
	RETURN;
END_IF

Base_Library.Tracing.Trace.Verbose(_MyName, 'Register Mover Accepted');
addMover.AddMover(MoverToAdd := MoverToAdd);
MoverToAdd.MyCAGroup  := THIS^;
FOR i := 0 TO MaxMovers DO
	IF GroupMovers[i] = 0 THEN
		GroupMovers[i] := MoverToAdd;
		RegisteredMovers := RegisteredMovers + 1;
		EXIT;
	END_IF
END_FOR
END_METHOD

PROPERTY AxisCount : UDINT
GET
AxisCount := _caGroup.NcToPlc.Common.GroupAxesCount;
END_GET
END_PROPERTY

PROPERTY CAGroupXtsIoEnvInterface : I_Mc2CaGroup
GET
CAGroupXtsIoEnvInterface := _ICaGroup;
END_GET
SET
_ICaGroup := CAGroupXtsIoEnvInterface;
IF _ICaGroup <> 0 THEN
	_MyName := _ICaGroup.P_ObjectName;
END_IF
END_SET
END_PROPERTY

METHOD Cycle : HRESULT
VAR
	ResetCaGroupResult : HRESULT;
	EnableCaGroupResult : HRESULT;
	DisableCaGroupResult : HRESULT;
	AddMoverCallResult: HRESULT;
	RemoveAllCycleResult: HRESULT;
	GrpStopCycleResult: HRESULT;
END_VAR
IF _ICaGroup = 0 THEN
	Cycle := -1;
	RETURN;
END_IF


ReadGroupStatus(AxesGroup:= _caGroup, Enable:= TRUE );
ReadErrorCode(AxesGroup := _caGroup, Enable := TRUE, GroupErrorId => GroupErrorCode);
ResetCaGroupResult := resetCAGroup.Cycle();
EnableCaGroupResult := enableCAGroup.Cycle();
DisableCaGroupResult := disableCAGroup.Cycle();
AddMoverCallResult := addMover.Cycle();
RemoveAllCycleResult := removeAllAxes.Cycle();
GrpStopCycleResult := grpStop.Cycle();
removeMover.Cycle();

//Cyclic get CaGroup information
stGroupInformation.sName := 'MainCAGroup';
stGroupInformation.eGroupState := _caGroup.NcToPlc.Common.GroupStatus.State;
stGroupInformation.nAxesCount	:= UDINT_TO_INT(_caGroup.NcToPlc.Common.GroupAxesCount);
stGroupInformation.nId			:= _caGroup.NcToPlc.Common.GroupOID;
END_METHOD

METHOD Disable : BOOL
VAR_INPUT
END_VAR
IF NOT disableCAGroup.Busy THEN
	Base_Library.Tracing.Trace.Verbose(_MyName, 'Group Disable Accepted');
	Disable := SUCCEEDED(disableCAGroup.Execute());
END_IF
END_METHOD

METHOD Enable : BOOL
VAR_INPUT
END_VAR
IF NOT enableCAGroup.Busy THEN
	Base_Library.Tracing.Trace.Verbose(_MyName, 'Group Enable Accepted');
	Enable := SUCCEEDED(enableCAGroup.Execute());
END_IF
END_METHOD

PROPERTY ErrorCode : UDINT
GET
ErrorCode := GroupErrorCode;
END_GET
END_PROPERTY

PROPERTY GroupRef : reference to AXES_GROUP_REF
GET
GroupRef REF= _caGroup;
END_GET
END_PROPERTY

METHOD GroupStop : BOOL
VAR_INPUT
END_VAR
IF NOT grpStop.Busy THEN
	Base_Library.Tracing.Trace.Verbose(_MyName, 'GroupStop accepted');
	GroupStop := SUCCEEDED(grpStop.Execute());
END_IF
END_METHOD

PROPERTY HasError : BOOL
GET
HasError := ReadGroupStatus.GroupErrorStop OR ReadGroupStatus.GroupNotReady;
END_GET
END_PROPERTY

PROPERTY IsDisabled : BOOL
GET
IsDisabled := ReadGroupStatus.GroupDisabled;
END_GET
END_PROPERTY

PROPERTY IsInErrorStop : BOOL
GET
IsInErrorStop := ReadGroupStatus.GroupErrorStop;
END_GET
END_PROPERTY

PROPERTY IsInStandBy : BOOL
GET
IsInStandBy := ReadGroupStatus.GroupStandby;
END_GET
END_PROPERTY

PROPERTY IsMoving : BOOL
GET
IsMoving := ReadGroupStatus.GroupMoving;
END_GET
END_PROPERTY

PROPERTY IsStopping : BOOL
GET
IsStopping := ReadGroupStatus.GroupStopping;
END_GET
END_PROPERTY

PROPERTY MyName : string
GET
MyName := _MyName;
END_GET
END_PROPERTY

METHOD RegisterWithParent
VAR_INPUT
	Parent	: I_HostObjects;
END_VAR
Parent.RegisterCyclic(THIS^);
END_METHOD

METHOD RemoveAllMovers : HRESULT
VAR
	i : INT;
END_VAR
IF removeAllAxes.Busy THEN
	Base_Library.Tracing.Trace.Warning(_MyName, 'Remove All Failed - busy');
	RemoveAllMovers := -1;
	RETURN;
END_IF
IF RegisteredMovers = 0 THEN
	Base_Library.Tracing.Trace.Warning(_MyName, 'Remove All Failed - No Movers');
	RemoveAllMovers := -2;
	RETURN;
END_IF

Base_Library.Tracing.Trace.Verbose(_MyName, 'Remove All Movers Accepted');
removeAllAxes.RemoveAllMover();
RegisteredMovers := 0;
FOR i := 0 TO MaxMovers DO
	GroupMovers[i] := 0;
END_FOR
END_METHOD

METHOD RemoveAMover : HRESULT
VAR_INPUT
	MoverToRemove : I_XtsMover;
END_VAR
VAR
	i : INT;
	registered : BOOL;
END_VAR
IF removeMover.Busy THEN
	Base_Library.Tracing.Trace.Warning(MyName, 'Remove Fail - busy');
	RemoveAMover := -1;
	RETURN;
END_IF
IF MoverToRemove = 0 THEN
	Base_Library.Tracing.Trace.Warning(MyName, 'Remove Fail - null ptr');
	RemoveAMover := -2;
	RETURN;
END_IF
FOR i := 0 TO MaxMovers DO
	IF GroupMovers[i] = MoverToRemove THEN
		registered := TRUE;
	END_IF
END_FOR
IF NOT registered THEN
	Base_Library.Tracing.Trace.Warning(MyName, 'Remove Fail - not registered');
	RemoveAMover := -2;
	RETURN;
END_IF

